LIN {X 0,Y 410.948,Z 878.716,A -85,B 0,C 180,E1 18093.627,E2 18093.627} C_VEL
LIN {X 0,Y 409.923,Z 893.274,A -85,B 0,C 180,E1 18092.657,E2 18092.657} C_VEL
LIN {X 0,Y 408.653,Z 907.82,A -85,B 0,C 180,E1 18091.402,E2 18091.402} C_VEL
LIN {X 0,Y 407.32,Z 921.375,A -85,B 0,C 180,E1 18089.93,E2 18089.93} C_VEL
LIN {X 0,Y 406.014,Z 933.316,A -85,B 0,C 180,E1 18088.307,E2 18088.307} C_VEL
LIN {X 0,Y 404.726,Z 944.345,A -85,B 0,C 180,E1 18086.441,E2 18086.441} C_VEL
LIN {X 0,Y 403.633,Z 953.739,A -85,B 0,C 180,E1 18084.456,E2 18084.456} C_VEL
LIN {X 0,Y 402.724,Z 961.665,A -85,B 0,C 180,E1 18082.296,E2 18082.296} C_VEL
LIN {X 0,Y 402.061,Z 968.085,A -85,B 0,C 180,E1 18079.975,E2 18079.975} C_VEL
LIN {X 0,Y 401.649,Z 972.603,A -85,B 0,C 180,E1 18077.638,E2 18077.638} C_VEL
LIN {X 0,Y 401.427,Z 975.501,A -85,B 0,C 180,E1 18075.11,E2 18075.11} C_VEL
LIN {X 0,Y 401.407,Z 976.508,A -85,B 0,C 180,E1 18072.758,E2 18072.758} C_VEL
LIN {X 0,Y 401.558,Z 975.728,A -85,B 0,C 180,E1 18070.255,E2 18070.255} C_VEL
LIN {X 0,Y 401.936,Z 973.165,A -85,B 0,C 180,E1 18067.783,E2 18067.783} C_VEL
LIN {X 0,Y 402.51,Z 969.039,A -85,B 0,C 180,E1 18065.491,E2 18065.491} C_VEL
LIN {X 0,Y 403.373,Z 962.973,A -85,B 0,C 180,E1 18063.171,E2 18063.171} C_VEL
LIN {X 0,Y 404.499,Z 955.48,A -85,B 0,C 180,E1 18061.022,E2 18061.022} C_VEL
LIN {X 0,Y 405.852,Z 946.406,A -85,B 0,C 180,E1 18059.01,E2 18059.01} C_VEL
LIN {X 0,Y 407.46,Z 935.302,A -85,B 0,C 180,E1 18057.059,E2 18057.059} C_VEL
LIN {X 0,Y 409.093,Z 923.229,A -85,B 0,C 180,E1 18055.365,E2 18055.365} C_VEL
LIN {X 0,Y 410.738,Z 909.55,A -85,B 0,C 180,E1 18053.843,E2 18053.843} C_VEL
LIN {X 0,Y 412.221,Z 895.286,A -85,B 0,C 180,E1 18052.584,E2 18052.584} C_VEL
LIN {X 0,Y 413.472,Z 880.507,A -85,B 0,C 180,E1 18051.576,E2 18051.576} C_VEL
LIN {X 0,Y 414.481,Z 863.966,A -85,B 0,C 180,E1 18050.742,E2 18050.742} C_VEL
LIN {X 0,Y 415.114,Z 847.179,A -85,B 0,C 180,E1 18050.169,E2 18050.169} C_VEL
LIN {X 0,Y 417.861,Z 722.491,A -85,B 0,C 180,E1 18047.832,E2 18047.832} C_VEL
LIN {X 0,Y 411.801,Z 695.607,A -85,B 0,C 180,E1 18046.697,E2 18046.697} C_VEL
LIN {X 0,Y 414.81,Z 668.603,A -85,B 0,C 180,E1 18042.474,E2 18042.474} C_VEL
LIN {X 0,Y 414.66,Z 666.207,A -85,B 0,C 180,E1 18042.041,E2 18042.041} C_VEL
LIN {X 0,Y 410.898,Z 651.984,A -85,B 0,C 180,E1 18039.068,E2 18039.068} C_VEL
LIN {X 0,Y 406.79,Z 639.122,A -85,B 0,C 180,E1 18036.151,E2 18036.151} C_VEL
LIN {X 0,Y 402.415,Z 627.066,A -85,B 0,C 180,E1 18033.142,E2 18033.142} C_VEL
LIN {X 0,Y 401.514,Z 624.334,A -85,B 0,C 180,E1 18032.371,E2 18032.371} C_VEL
LIN {X 0,Y 401.502,Z 624.212,A -85,B 0,C 180,E1 18028.402,E2 18028.402} C_VEL
LIN {X 0,Y 401.498,Z 624.219,A -85,B 0,C 180,E1 18024.419,E2 18024.419} C_VEL
LIN {X 0,Y 401.497,Z 624.224,A -85,B 0,C 180,E1 18020.405,E2 18020.405} C_VEL
LIN {X 0,Y 401.498,Z 624.224,A -85,B 0,C 180,E1 18016.344,E2 18016.344} C_VEL
LIN {X 0,Y 401.501,Z 624.222,A -85,B 0,C 180,E1 18012.367,E2 18012.367} C_VEL
LIN {X 0,Y 401.501,Z 624.22,A -85,B 0,C 180,E1 18008.305,E2 18008.305} C_VEL
LIN {X 0,Y 401.491,Z 624.213,A -85,B 0,C 180,E1 18004.428,E2 18004.428} C_VEL
LIN {X 0,Y 401.485,Z 624.204,A -85,B 0,C 180,E1 18000.428,E2 18000.428} C_VEL
LIN {X 0,Y 401.482,Z 624.205,A -85,B 0,C 180,E1 17996.431,E2 17996.431} C_VEL
LIN {X 0,Y 401.486,Z 624.215,A -85,B 0,C 180,E1 17992.416,E2 17992.416} C_VEL
LIN {X 0,Y 401.494,Z 624.224,A -85,B 0,C 180,E1 17988.508,E2 17988.508} C_VEL
LIN {X 0,Y 401.5,Z 624.215,A -85,B 0,C 180,E1 17984.525,E2 17984.525} C_VEL
LIN {X 0,Y 401.5,Z 624.206,A -85,B 0,C 180,E1 17980.507,E2 17980.507} C_VEL
LIN {X 0,Y 401.501,Z 624.205,A -85,B 0,C 180,E1 17976.519,E2 17976.519} C_VEL
LIN {X 0,Y 401.501,Z 624.206,A -85,B 0,C 180,E1 17972.568,E2 17972.568} C_VEL
LIN {X 0,Y 401.5,Z 624.207,A -85,B 0,C 180,E1 17968.636,E2 17968.636} C_VEL
LIN {X 0,Y 401.486,Z 624.213,A -85,B 0,C 180,E1 17964.706,E2 17964.706} C_VEL
LIN {X 0,Y 401.479,Z 624.224,A -85,B 0,C 180,E1 17960.76,E2 17960.76} C_VEL
LIN {X 0,Y 401.478,Z 624.222,A -85,B 0,C 180,E1 17956.775,E2 17956.775} C_VEL
LIN {X 0,Y 401.58,Z 624.794,A -85,B 0,C 180,E1 17956.338,E2 17956.338} C_VEL
LIN {X 0,Y 406.93,Z 637.442,A -85,B 0,C 180,E1 17953.665,E2 17953.665} C_VEL
LIN {X 0,Y 412.612,Z 651.727,A -85,B 0,C 180,E1 17950.989,E2 17950.989} C_VEL
LIN {X 0,Y 417.899,Z 667.344,A -85,B 0,C 180,E1 17948.423,E2 17948.423} C_VEL
LIN {X 0,Y 419.949,Z 674.277,A -85,B 0,C 180,E1 17947.382,E2 17947.382} C_VEL
LIN {X 0,Y 416.011,Z 707.311,A -85,B 0,C 180,E1 17943.954,E2 17943.954} C_VEL
LIN {X 0,Y 419.913,Z 739.224,A -85,B 0,C 180,E1 17942.952,E2 17942.952} C_VEL
LIN {X 0,Y 415.985,Z 917.427,A -85,B 0,C 180,E1 17939.753,E2 17939.753} C_VEL
LIN {X 0,Y 414.846,Z 936.641,A -85,B 0,C 180,E1 17939.174,E2 17939.174} C_VEL
LIN {X 0,Y 413.402,Z 954.824,A -85,B 0,C 180,E1 17938.376,E2 17938.376} C_VEL
LIN {X 0,Y 411.674,Z 972.774,A -85,B 0,C 180,E1 17937.325,E2 17937.325} C_VEL
LIN {X 0,Y 409.84,Z 989.883,A -85,B 0,C 180,E1 17936.048,E2 17936.048} C_VEL
LIN {X 0,Y 407.953,Z 1006.197,A -85,B 0,C 180,E1 17934.546,E2 17934.546} C_VEL
LIN {X 0,Y 406.111,Z 1021.663,A -85,B 0,C 180,E1 17932.815,E2 17932.815} C_VEL
LIN {X 0,Y 404.421,Z 1036.236,A -85,B 0,C 180,E1 17930.847,E2 17930.847} C_VEL
LIN {X 0,Y 402.954,Z 1049.621,A -85,B 0,C 180,E1 17928.668,E2 17928.668} C_VEL
LIN {X 0,Y 401.838,Z 1061.521,A -85,B 0,C 180,E1 17926.33,E2 17926.33} C_VEL
LIN {X 0,Y 401.058,Z 1071.88,A -85,B 0,C 180,E1 17923.847,E2 17923.847} C_VEL
LIN {X 0,Y 400.626,Z 1080.6,A -85,B 0,C 180,E1 17921.239,E2 17921.239} C_VEL
LIN {X 0,Y 400.459,Z 1087.386,A -85,B 0,C 180,E1 17918.613,E2 17918.613} C_VEL
LIN {X 0,Y 400.468,Z 1092.26,A -85,B 0,C 180,E1 17916.019,E2 17916.019} C_VEL
LIN {X 0,Y 400.552,Z 1095.388,A -85,B 0,C 180,E1 17913.434,E2 17913.434} C_VEL
LIN {X 0,Y 400.609,Z 1096.821,A -85,B 0,C 180,E1 17910.858,E2 17910.858} C_VEL
LIN {X 0,Y 400.591,Z 1096.647,A -85,B 0,C 180,E1 17908.426,E2 17908.426} C_VEL
LIN {X 0,Y 400.513,Z 1094.819,A -85,B 0,C 180,E1 17905.848,E2 17905.848} C_VEL
LIN {X 0,Y 400.431,Z 1091.265,A -85,B 0,C 180,E1 17903.26,E2 17903.26} C_VEL
LIN {X 0,Y 400.461,Z 1085.91,A -85,B 0,C 180,E1 17900.66,E2 17900.66} C_VEL
LIN {X 0,Y 400.699,Z 1078.507,A -85,B 0,C 180,E1 17898.001,E2 17898.001} C_VEL
LIN {X 0,Y 401.246,Z 1069.273,A -85,B 0,C 180,E1 17895.423,E2 17895.423} C_VEL
LIN {X 0,Y 402.084,Z 1058.931,A -85,B 0,C 180,E1 17893.085,E2 17893.085} C_VEL
LIN {X 0,Y 403.252,Z 1046.965,A -85,B 0,C 180,E1 17890.854,E2 17890.854} C_VEL
LIN {X 0,Y 404.735,Z 1033.331,A -85,B 0,C 180,E1 17888.749,E2 17888.749} C_VEL
LIN {X 0,Y 406.383,Z 1018.854,A -85,B 0,C 180,E1 17886.894,E2 17886.894} C_VEL
LIN {X 0,Y 408.163,Z 1003.233,A -85,B 0,C 180,E1 17885.235,E2 17885.235} C_VEL
LIN {X 0,Y 409.958,Z 986.785,A -85,B 0,C 180,E1 17883.803,E2 17883.803} C_VEL
LIN {X 0,Y 411.678,Z 969.565,A -85,B 0,C 180,E1 17882.597,E2 17882.597} C_VEL
LIN {X 0,Y 413.244,Z 951.519,A -85,B 0,C 180,E1 17881.612,E2 17881.612} C_VEL
LIN {X 0,Y 414.584,Z 932.755,A -85,B 0,C 180,E1 17880.86,E2 17880.86} C_VEL
LIN {X 0,Y 415.491,Z 913.481,A -85,B 0,C 180,E1 17880.346,E2 17880.346} C_VEL
LIN {X 0,Y 418.723,Z 737.102,A -85,B 0,C 180,E1 17877.259,E2 17877.259} C_VEL
LIN {X 0,Y 414.963,Z 707.158,A -85,B 0,C 180,E1 17876.389,E2 17876.389} C_VEL
LIN {X 0,Y 418.463,Z 672.256,A -85,B 0,C 180,E1 17872.887,E2 17872.887} C_VEL
LIN {X 0,Y 411.146,Z 650.69,A -85,B 0,C 180,E1 17869.783,E2 17869.783} C_VEL
LIN {X 0,Y 403.769,Z 630.541,A -85,B 0,C 180,E1 17866.618,E2 17866.618} C_VEL
LIN {X 0,Y 401.517,Z 624.406,A -85,B 0,C 180,E1 17865.527,E2 17865.527} C_VEL
LIN {X 0,Y 401.497,Z 624.217,A -85,B 0,C 180,E1 17861.66,E2 17861.66} C_VEL
LIN {X 0,Y 401.499,Z 624.222,A -85,B 0,C 180,E1 17857.779,E2 17857.779} C_VEL
LIN {X 0,Y 401.492,Z 624.224,A -85,B 0,C 180,E1 17853.906,E2 17853.906} C_VEL
LIN {X 0,Y 401.484,Z 624.224,A -85,B 0,C 180,E1 17849.926,E2 17849.926} C_VEL
LIN {X 0,Y 401.483,Z 624.224,A -85,B 0,C 180,E1 17845.967,E2 17845.967} C_VEL
LIN {X 0,Y 401.488,Z 624.225,A -85,B 0,C 180,E1 17842.089,E2 17842.089} C_VEL
LIN {X 0,Y 401.49,Z 624.226,A -85,B 0,C 180,E1 17838.137,E2 17838.137} C_VEL
LIN {X 0,Y 401.509,Z 624.334,A -85,B 0,C 180,E1 17834.714,E2 17834.714} C_VEL
LIN {X 0,Y 402.009,Z 626.178,A -85,B 0,C 180,E1 17834.328,E2 17834.328} C_VEL
LIN {X 0,Y 406.281,Z 636.393,A -85,B 0,C 180,E1 17832.58,E2 17832.58} C_VEL
LIN {X 0,Y 410.796,Z 649.556,A -85,B 0,C 180,E1 17830.518,E2 17830.518} C_VEL
LIN {X 0,Y 413.885,Z 662.108,A -85,B 0,C 180,E1 17828.684,E2 17828.684} C_VEL
LIN {X 0,Y 413.166,Z 694.495,A -85,B 0,C 180,E1 17824.859,E2 17824.859} C_VEL
LIN {X 0,Y 412.587,Z 720.52,A -85,B 0,C 180,E1 17821.757,E2 17821.757} C_VEL
LIN {X 0,Y 412.786,Z 724.532,A -85,B 0,C 180,E1 17821.644,E2 17821.644} C_VEL
LIN {X 0,Y 409.599,Z 849.624,A -85,B 0,C 180,E1 17819.025,E2 17819.025} C_VEL
LIN {X 0,Y 409.503,Z 867.341,A -85,B 0,C 180,E1 17818.522,E2 17818.522} C_VEL
LIN {X 0,Y 409.073,Z 883.957,A -85,B 0,C 180,E1 17817.758,E2 17817.758} C_VEL
LIN {X 0,Y 408.449,Z 898.379,A -85,B 0,C 180,E1 17816.842,E2 17816.842} C_VEL
LIN {X 0,Y 407.57,Z 912.742,A -85,B 0,C 180,E1 17815.638,E2 17815.638} C_VEL
LIN {X 0,Y 406.631,Z 925.44,A -85,B 0,C 180,E1 17814.284,E2 17814.284} C_VEL
LIN {X 0,Y 405.541,Z 937.675,A -85,B 0,C 180,E1 17812.634,E2 17812.634} C_VEL
LIN {X 0,Y 404.547,Z 947.904,A -85,B 0,C 180,E1 17810.898,E2 17810.898} C_VEL
LIN {X 0,Y 403.573,Z 957.408,A -85,B 0,C 180,E1 17808.844,E2 17808.844} C_VEL
LIN {X 0,Y 402.819,Z 964.607,A -85,B 0,C 180,E1 17806.799,E2 17806.799} C_VEL
LIN {X 0,Y 402.216,Z 970.369,A -85,B 0,C 180,E1 17804.574,E2 17804.574} C_VEL
LIN {X 0,Y 401.791,Z 974.195,A -85,B 0,C 180,E1 17802.326,E2 17802.326} C_VEL
LIN {X 0,Y 401.543,Z 976.273,A -85,B 0,C 180,E1 17800.054,E2 17800.054} C_VEL
LIN {X 0,Y 401.425,Z 976.558,A -85,B 0,C 180,E1 17797.753,E2 17797.753} C_VEL
LIN {X 0,Y 401.434,Z 975.029,A -85,B 0,C 180,E1 17795.384,E2 17795.384} C_VEL
LIN {X 0,Y 401.568,Z 971.912,A -85,B 0,C 180,E1 17793.213,E2 17793.213} C_VEL
LIN {X 0,Y 401.869,Z 966.938,A -85,B 0,C 180,E1 17790.976,E2 17790.976} C_VEL
LIN {X 0,Y 402.325,Z 960.411,A -85,B 0,C 180,E1 17788.874,E2 17788.874} C_VEL
LIN {X 0,Y 402.989,Z 951.677,A -85,B 0,C 180,E1 17786.735,E2 17786.735} C_VEL
LIN {X 0,Y 403.732,Z 942.257,A -85,B 0,C 180,E1 17784.931,E2 17784.931} C_VEL
LIN {X 0,Y 404.673,Z 930.317,A -85,B 0,C 180,E1 17783.101,E2 17783.101} C_VEL
LIN {X 0,Y 405.573,Z 917.892,A -85,B 0,C 180,E1 17781.592,E2 17781.592} C_VEL
LIN {X 0,Y 406.458,Z 904.008,A -85,B 0,C 180,E1 17780.239,E2 17780.239} C_VEL
LIN {X 0,Y 407.25,Z 888.689,A -85,B 0,C 180,E1 17779.089,E2 17779.089} C_VEL
LIN {X 0,Y 407.854,Z 873.417,A -85,B 0,C 180,E1 17778.225,E2 17778.225} C_VEL
LIN {X 0,Y 408.225,Z 856.157,A -85,B 0,C 180,E1 17777.554,E2 17777.554} C_VEL
LIN {X 0,Y 408.39,Z 834.696,A -85,B 0,C 180,E1 17777.069,E2 17777.069} C_VEL
LIN {X 0,Y 410.575,Z 718.657,A -85,B 0,C 180,E1 17774.8,E2 17774.8} C_VEL
LIN {X 0,Y 409.2,Z 710.904,A -85,B 0,C 180,E1 17774.53,E2 17774.53} C_VEL
LIN {X 0,Y 410.192,Z 680.126,A -85,B 0,C 180,E1 17770.705,E2 17770.705} C_VEL
LIN {X 0,Y 410.726,Z 657.174,A -85,B 0,C 180,E1 17767.841,E2 17767.841} C_VEL
LIN {X 0,Y 405.666,Z 638.159,A -85,B 0,C 180,E1 17765.05,E2 17765.05} C_VEL
LIN {X 0,Y 401.475,Z 624.396,A -85,B 0,C 180,E1 17762.912,E2 17762.912} C_VEL
LIN {X 0,Y 401.489,Z 624.225,A -85,B 0,C 180,E1 17761.35,E2 17761.35} C_VEL
LIN {X 0,Y 400.432,Z 624.354,A -85,B 0,C 180,E1 17760.251,E2 17760.251} C_VEL
LIN {X 0,Y 393.938,Z 625.162,A -85,B 0,C 180,E1 17757.072,E2 17757.072} C_VEL
LIN {X 0,Y 393.509,Z 625.198,A -85,B 0,C 180,E1 17756.342,E2 17756.342} C_VEL
LIN {X 0,Y 393.515,Z 625.213,A -85,B 0,C 180,E1 17752.351,E2 17752.351} C_VEL
LIN {X 0,Y 393.611,Z 625.529,A -85,B 0,C 180,E1 17751.144,E2 17751.144} C_VEL
LIN {X 0,Y 398.734,Z 642.233,A -85,B 0,C 180,E1 17747.657,E2 17747.657} C_VEL
LIN {X 0,Y 403.375,Z 659.305,A -85,B 0,C 180,E1 17744.352,E2 17744.352} C_VEL
LIN {X 0,Y 404.657,Z 665.567,A -85,B 0,C 180,E1 17743.211,E2 17743.211} C_VEL
LIN {X 0,Y 401.936,Z 693.579,A -85,B 0,C 180,E1 17738.873,E2 17738.873} C_VEL
LIN {X 0,Y 401.915,Z 695.836,A -85,B 0,C 180,E1 17738.621,E2 17738.621} C_VEL
LIN {X 0,Y 407.444,Z 724.144,A -85,B 0,C 180,E1 17737.677,E2 17737.677} C_VEL
LIN {X 0,Y 404.979,Z 846.669,A -85,B 0,C 180,E1 17735.424,E2 17735.424} C_VEL
LIN {X 0,Y 404.395,Z 863.875,A -85,B 0,C 180,E1 17734.831,E2 17734.831} C_VEL
LIN {X 0,Y 403.562,Z 879.387,A -85,B 0,C 180,E1 17734.049,E2 17734.049} C_VEL
LIN {X 0,Y 402.492,Z 894.012,A -85,B 0,C 180,E1 17733.062,E2 17733.062} C_VEL
LIN {X 0,Y 401.135,Z 908.873,A -85,B 0,C 180,E1 17731.759,E2 17731.759} C_VEL
LIN {X 0,Y 399.76,Z 922.197,A -85,B 0,C 180,E1 17730.287,E2 17730.287} C_VEL
LIN {X 0,Y 398.444,Z 933.729,A -85,B 0,C 180,E1 17728.706,E2 17728.706} C_VEL
LIN {X 0,Y 397.085,Z 944.773,A -85,B 0,C 180,E1 17726.825,E2 17726.825} C_VEL
LIN {X 0,Y 395.904,Z 954.369,A -85,B 0,C 180,E1 17724.784,E2 17724.784} C_VEL
LIN {X 0,Y 394.99,Z 961.973,A -85,B 0,C 180,E1 17722.729,E2 17722.729} C_VEL
LIN {X 0,Y 394.252,Z 968.582,A -85,B 0,C 180,E1 17720.365,E2 17720.365} C_VEL
LIN {X 0,Y 393.789,Z 973.345,A -85,B 0,C 180,E1 17717.983,E2 17717.983} C_VEL
LIN {X 0,Y 393.539,Z 976.31,A -85,B 0,C 180,E1 17715.583,E2 17715.583} C_VEL
LIN {X 0,Y 393.487,Z 977.642,A -85,B 0,C 180,E1 17713.01,E2 17713.01} C_VEL
LIN {X 0,Y 393.631,Z 977.211,A -85,B 0,C 180,E1 17710.564,E2 17710.564} C_VEL
LIN {X 0,Y 393.986,Z 974.982,A -85,B 0,C 180,E1 17708.096,E2 17708.096} C_VEL
LIN {X 0,Y 394.603,Z 970.926,A -85,B 0,C 180,E1 17705.606,E2 17705.606} C_VEL
LIN {X 0,Y 395.488,Z 965.214,A -85,B 0,C 180,E1 17703.256,E2 17703.256} C_VEL
LIN {X 0,Y 396.743,Z 957.38,A -85,B 0,C 180,E1 17700.897,E2 17700.897} C_VEL
LIN {X 0,Y 398.171,Z 948.589,A -85,B 0,C 180,E1 17698.85,E2 17698.85} C_VEL
LIN {X 0,Y 399.806,Z 937.996,A -85,B 0,C 180,E1 17696.908,E2 17696.908} C_VEL
LIN {X 0,Y 401.524,Z 926.181,A -85,B 0,C 180,E1 17695.169,E2 17695.169} C_VEL
LIN {X 0,Y 403.213,Z 913.39,A -85,B 0,C 180,E1 17693.655,E2 17693.655} C_VEL
LIN {X 0,Y 404.818,Z 899.074,A -85,B 0,C 180,E1 17692.317,E2 17692.317} C_VEL
LIN {X 0,Y 406.277,Z 883.536,A -85,B 0,C 180,E1 17691.187,E2 17691.187} C_VEL
LIN {X 0,Y 407.372,Z 867.647,A -85,B 0,C 180,E1 17690.329,E2 17690.329} C_VEL
LIN {X 0,Y 408.106,Z 850.469,A -85,B 0,C 180,E1 17689.693,E2 17689.693} C_VEL
LIN {X 0,Y 408.732,Z 823.466,A -85,B 0,C 180,E1 17689.121,E2 17689.121} C_VEL
LIN {X 0,Y 411.102,Z 723.877,A -85,B 0,C 180,E1 17687.253,E2 17687.253} C_VEL
LIN {X 0,Y 404.768,Z 695.985,A -85,B 0,C 180,E1 17686.043,E2 17686.043} C_VEL
LIN {X 0,Y 407.748,Z 670.492,A -85,B 0,C 180,E1 17682.013,E2 17682.013} C_VEL
LIN {X 0,Y 404.253,Z 656.746,A -85,B 0,C 180,E1 17679.103,E2 17679.103} C_VEL
LIN {X 0,Y 400.252,Z 643.813,A -85,B 0,C 180,E1 17676.125,E2 17676.125} C_VEL
LIN {X 0,Y 395.853,Z 631.559,A -85,B 0,C 180,E1 17673.01,E2 17673.01} C_VEL
LIN {X 0,Y 393.578,Z 625.315,A -85,B 0,C 180,E1 17671.253,E2 17671.253} C_VEL
LIN {X 0,Y 393.565,Z 625.213,A -85,B 0,C 180,E1 17667.213,E2 17667.213} C_VEL
LIN {X 0,Y 393.561,Z 625.205,A -85,B 0,C 180,E1 17663.122,E2 17663.122} C_VEL
LIN {X 0,Y 393.556,Z 625.199,A -85,B 0,C 180,E1 17659.075,E2 17659.075} C_VEL
LIN {X 0,Y 393.549,Z 625.199,A -85,B 0,C 180,E1 17655.109,E2 17655.109} C_VEL
LIN {X 0,Y 393.55,Z 625.202,A -85,B 0,C 180,E1 17651.133,E2 17651.133} C_VEL
LIN {X 0,Y 393.555,Z 625.208,A -85,B 0,C 180,E1 17647.152,E2 17647.152} C_VEL
LIN {X 0,Y 393.557,Z 625.214,A -85,B 0,C 180,E1 17643.201,E2 17643.201} C_VEL
LIN {X 0,Y 393.562,Z 625.203,A -85,B 0,C 180,E1 17639.127,E2 17639.127} C_VEL
LIN {X 0,Y 393.558,Z 625.19,A -85,B 0,C 180,E1 17635.045,E2 17635.045} C_VEL
LIN {X 0,Y 393.559,Z 625.189,A -85,B 0,C 180,E1 17631.085,E2 17631.085} C_VEL
LIN {X 0,Y 393.56,Z 625.198,A -85,B 0,C 180,E1 17627.082,E2 17627.082} C_VEL
LIN {X 0,Y 393.562,Z 625.211,A -85,B 0,C 180,E1 17623.165,E2 17623.165} C_VEL
LIN {X 0,Y 393.56,Z 625.211,A -85,B 0,C 180,E1 17619.165,E2 17619.165} C_VEL
LIN {X 0,Y 393.549,Z 625.212,A -85,B 0,C 180,E1 17615.216,E2 17615.216} C_VEL
LIN {X 0,Y 393.545,Z 625.211,A -85,B 0,C 180,E1 17611.225,E2 17611.225} C_VEL
LIN {X 0,Y 393.543,Z 625.214,A -85,B 0,C 180,E1 17607.238,E2 17607.238} C_VEL
LIN {X 0,Y 393.547,Z 625.214,A -85,B 0,C 180,E1 17603.341,E2 17603.341} C_VEL
LIN {X 0,Y 393.561,Z 625.203,A -85,B 0,C 180,E1 17599.43,E2 17599.43} C_VEL
LIN {X 0,Y 393.6,Z 625.474,A -85,B 0,C 180,E1 17597.551,E2 17597.551} C_VEL
LIN {X 0,Y 398.76,Z 637.635,A -85,B 0,C 180,E1 17594.796,E2 17594.796} C_VEL
LIN {X 0,Y 404.277,Z 651.337,A -85,B 0,C 180,E1 17592.085,E2 17592.085} C_VEL
LIN {X 0,Y 409.518,Z 666.021,A -85,B 0,C 180,E1 17589.509,E2 17589.509} C_VEL
LIN {X 0,Y 412.843,Z 677.235,A -85,B 0,C 180,E1 17587.743,E2 17587.743} C_VEL
LIN {X 0,Y 409.049,Z 707.569,A -85,B 0,C 180,E1 17584.547,E2 17584.547} C_VEL
LIN {X 0,Y 413.042,Z 740.309,A -85,B 0,C 180,E1 17583.504,E2 17583.504} C_VEL
LIN {X 0,Y 408.913,Z 916.579,A -85,B 0,C 180,E1 17580.285,E2 17580.285} C_VEL
LIN {X 0,Y 407.728,Z 935.734,A -85,B 0,C 180,E1 17579.699,E2 17579.699} C_VEL
LIN {X 0,Y 406.253,Z 953.317,A -85,B 0,C 180,E1 17578.922,E2 17578.922} C_VEL
LIN {X 0,Y 404.435,Z 971.385,A -85,B 0,C 180,E1 17577.856,E2 17577.856} C_VEL
LIN {X 0,Y 402.486,Z 988.565,A -85,B 0,C 180,E1 17576.561,E2 17576.561} C_VEL
LIN {X 0,Y 400.472,Z 1004.977,A -85,B 0,C 180,E1 17575.028,E2 17575.028} C_VEL
LIN {X 0,Y 398.525,Z 1020.37,A -85,B 0,C 180,E1 17573.275,E2 17573.275} C_VEL
LIN {X 0,Y 396.728,Z 1034.89,A -85,B 0,C 180,E1 17571.279,E2 17571.279} C_VEL
LIN {X 0,Y 395.252,Z 1047.548,A -85,B 0,C 180,E1 17569.199,E2 17569.199} C_VEL
LIN {X 0,Y 394.023,Z 1059.595,A -85,B 0,C 180,E1 17566.815,E2 17566.815} C_VEL
LIN {X 0,Y 393.162,Z 1070.08,A -85,B 0,C 180,E1 17564.281,E2 17564.281} C_VEL
LIN {X 0,Y 392.68,Z 1078.97,A -85,B 0,C 180,E1 17561.604,E2 17561.604} C_VEL
LIN {X 0,Y 392.504,Z 1085.837,A -85,B 0,C 180,E1 17558.939,E2 17558.939} C_VEL
LIN {X 0,Y 392.519,Z 1090.833,A -85,B 0,C 180,E1 17556.288,E2 17556.288} C_VEL
LIN {X 0,Y 392.622,Z 1094.07,A -85,B 0,C 180,E1 17553.65,E2 17553.65} C_VEL
LIN {X 0,Y 392.694,Z 1095.604,A -85,B 0,C 180,E1 17551.021,E2 17551.021} C_VEL
LIN {X 0,Y 392.678,Z 1095.522,A -85,B 0,C 180,E1 17548.541,E2 17548.541} C_VEL
LIN {X 0,Y 392.59,Z 1093.764,A -85,B 0,C 180,E1 17545.91,E2 17545.91} C_VEL
LIN {X 0,Y 392.492,Z 1090.261,A -85,B 0,C 180,E1 17543.27,E2 17543.27} C_VEL
LIN {X 0,Y 392.504,Z 1084.969,A -85,B 0,C 180,E1 17540.617,E2 17540.617} C_VEL
LIN {X 0,Y 392.707,Z 1078.215,A -85,B 0,C 180,E1 17538.098,E2 17538.098} C_VEL
LIN {X 0,Y 393.204,Z 1069.612,A -85,B 0,C 180,E1 17535.569,E2 17535.569} C_VEL
LIN {X 0,Y 394.026,Z 1059.571,A -85,B 0,C 180,E1 17533.185,E2 17533.185} C_VEL
LIN {X 0,Y 395.163,Z 1048.166,A -85,B 0,C 180,E1 17530.949,E2 17530.949} C_VEL
LIN {X 0,Y 396.657,Z 1034.941,A -85,B 0,C 180,E1 17528.794,E2 17528.794} C_VEL
LIN {X 0,Y 398.417,Z 1020.149,A -85,B 0,C 180,E1 17526.796,E2 17526.796} C_VEL
LIN {X 0,Y 400.323,Z 1004.299,A -85,B 0,C 180,E1 17525.032,E2 17525.032} C_VEL
LIN {X 0,Y 402.243,Z 987.624,A -85,B 0,C 180,E1 17523.522,E2 17523.522} C_VEL
LIN {X 0,Y 404.046,Z 970.475,A -85,B 0,C 180,E1 17522.275,E2 17522.275} C_VEL
LIN {X 0,Y 405.725,Z 952.163,A -85,B 0,C 180,E1 17521.238,E2 17521.238} C_VEL
LIN {X 0,Y 407.153,Z 933.246,A -85,B 0,C 180,E1 17520.451,E2 17520.451} C_VEL
LIN {X 0,Y 408.129,Z 914.052,A -85,B 0,C 180,E1 17519.916,E2 17519.916} C_VEL
LIN {X 0,Y 411.541,Z 738.121,A -85,B 0,C 180,E1 17516.783,E2 17516.783} C_VEL
LIN {X 0,Y 407.676,Z 707.337,A -85,B 0,C 180,E1 17515.894,E2 17515.894} C_VEL
LIN {X 0,Y 411.164,Z 675.114,A -85,B 0,C 180,E1 17512.607,E2 17512.607} C_VEL
LIN {X 0,Y 404.132,Z 654.184,A -85,B 0,C 180,E1 17509.544,E2 17509.544} C_VEL
LIN {X 0,Y 397.156,Z 634.971,A -85,B 0,C 180,E1 17506.473,E2 17506.473} C_VEL
LIN {X 0,Y 393.584,Z 625.393,A -85,B 0,C 180,E1 17504.766,E2 17504.766} C_VEL
LIN {X 0,Y 393.567,Z 625.208,A -85,B 0,C 180,E1 17500.761,E2 17500.761} C_VEL
LIN {X 0,Y 393.561,Z 625.211,A -85,B 0,C 180,E1 17496.839,E2 17496.839} C_VEL
LIN {X 0,Y 393.56,Z 625.211,A -85,B 0,C 180,E1 17492.761,E2 17492.761} C_VEL
LIN {X 0,Y 393.569,Z 625.212,A -85,B 0,C 180,E1 17488.695,E2 17488.695} C_VEL
LIN {X 0,Y 393.566,Z 625.211,A -85,B 0,C 180,E1 17484.623,E2 17484.623} C_VEL
LIN {X 0,Y 393.569,Z 625.212,A -85,B 0,C 180,E1 17480.679,E2 17480.679} C_VEL
LIN {X 0,Y 393.561,Z 625.213,A -85,B 0,C 180,E1 17476.683,E2 17476.683} C_VEL
LIN {X 0,Y 393.565,Z 625.482,A -85,B 0,C 180,E1 17475.622,E2 17475.622} C_VEL
LIN {X 0,Y 394.9,Z 628.784,A -85,B 0,C 180,E1 17474.966,E2 17474.966} C_VEL
LIN {X 0,Y 400.239,Z 641.697,A -85,B 0,C 180,E1 17472.699,E2 17472.699} C_VEL
LIN {X 0,Y 404.726,Z 655.471,A -85,B 0,C 180,E1 17470.501,E2 17470.501} C_VEL
LIN {X 0,Y 406.969,Z 665.302,A -85,B 0,C 180,E1 17469.046,E2 17469.046} C_VEL
LIN {X 0,Y 406.169,Z 696.789,A -85,B 0,C 180,E1 17465.296,E2 17465.296} C_VEL
LIN {X 0,Y 405.53,Z 721.985,A -85,B 0,C 180,E1 17462.269,E2 17462.269} C_VEL
LIN {X 0,Y 405.725,Z 725.942,A -85,B 0,C 180,E1 17462.154,E2 17462.154} C_VEL
LIN {X 0,Y 402.305,Z 847.525,A -85,B 0,C 180,E1 17459.537,E2 17459.537} C_VEL
LIN {X 0,Y 402.217,Z 866.083,A -85,B 0,C 180,E1 17459.038,E2 17459.038} C_VEL
LIN {X 0,Y 401.86,Z 881.788,A -85,B 0,C 180,E1 17458.36,E2 17458.36} C_VEL
LIN {X 0,Y 401.192,Z 896.972,A -85,B 0,C 180,E1 17457.429,E2 17457.429} C_VEL
LIN {X 0,Y 400.326,Z 911.218,A -85,B 0,C 180,E1 17456.276,E2 17456.276} C_VEL
LIN {X 0,Y 399.259,Z 925.079,A -85,B 0,C 180,E1 17454.827,E2 17454.827} C_VEL
LIN {X 0,Y 398.245,Z 936.232,A -85,B 0,C 180,E1 17453.368,E2 17453.368} C_VEL
LIN {X 0,Y 397.141,Z 946.99,A -85,B 0,C 180,E1 17451.603,E2 17451.603} C_VEL
LIN {X 0,Y 396.127,Z 956.316,A -85,B 0,C 180,E1 17449.676,E2 17449.676} C_VEL
LIN {X 0,Y 395.235,Z 964.19,A -85,B 0,C 180,E1 17447.556,E2 17447.556} C_VEL
LIN {X 0,Y 394.578,Z 970.034,A -85,B 0,C 180,E1 17445.465,E2 17445.465} C_VEL
LIN {X 0,Y 394.052,Z 974.431,A -85,B 0,C 180,E1 17443.186,E2 17443.186} C_VEL
LIN {X 0,Y 393.724,Z 977.083,A -85,B 0,C 180,E1 17440.856,E2 17440.856} C_VEL
LIN {X 0,Y 393.544,Z 977.893,A -85,B 0,C 180,E1 17438.417,E2 17438.417} C_VEL
LIN {X 0,Y 393.508,Z 976.962,A -85,B 0,C 180,E1 17436.167,E2 17436.167} C_VEL
LIN {X 0,Y 393.612,Z 974.05,A -85,B 0,C 180,E1 17433.728,E2 17433.728} C_VEL
LIN {X 0,Y 393.886,Z 969.49,A -85,B 0,C 180,E1 17431.439,E2 17431.439} C_VEL
LIN {X 0,Y 394.345,Z 963.075,A -85,B 0,C 180,E1 17429.191,E2 17429.191} C_VEL
LIN {X 0,Y 394.928,Z 955.554,A -85,B 0,C 180,E1 17427.194,E2 17427.194} C_VEL
LIN {X 0,Y 395.764,Z 945.394,A -85,B 0,C 180,E1 17425.094,E2 17425.094} C_VEL
LIN {X 0,Y 396.657,Z 934.498,A -85,B 0,C 180,E1 17423.315,E2 17423.315} C_VEL
LIN {X 0,Y 397.679,Z 921.432,A -85,B 0,C 180,E1 17421.609,E2 17421.609} C_VEL
LIN {X 0,Y 398.576,Z 908.058,A -85,B 0,C 180,E1 17420.231,E2 17420.231} C_VEL
LIN {X 0,Y 399.44,Z 893.131,A -85,B 0,C 180,E1 17419.017,E2 17419.017} C_VEL
LIN {X 0,Y 400.124,Z 877.239,A -85,B 0,C 180,E1 17418.052,E2 17418.052} C_VEL
LIN {X 0,Y 400.56,Z 861.087,A -85,B 0,C 180,E1 17417.352,E2 17417.352} C_VEL
LIN {X 0,Y 400.731,Z 842.468,A -85,B 0,C 180,E1 17416.863,E2 17416.863} C_VEL
LIN {X 0,Y 403.114,Z 719.67,A -85,B 0,C 180,E1 17414.398,E2 17414.398} C_VEL
LIN {X 0,Y 401.725,Z 711.979,A -85,B 0,C 180,E1 17414.137,E2 17414.137} C_VEL
LIN {X 0,Y 402.764,Z 681.31,A -85,B 0,C 180,E1 17410.302,E2 17410.302} C_VEL
LIN {X 0,Y 403.271,Z 659.615,A -85,B 0,C 180,E1 17407.585,E2 17407.585} C_VEL
LIN {X 0,Y 398.366,Z 641.115,A -85,B 0,C 180,E1 17404.841,E2 17404.841} C_VEL
LIN {X 0,Y 393.534,Z 625.4,A -85,B 0,C 180,E1 17402.377,E2 17402.377} C_VEL
LIN {X 0,Y 393.51,Z 625.214,A -85,B 0,C 180,E1 17398.369,E2 17398.369} C_VEL
LIN {X 0,Y 393.509,Z 625.198,A -85,B 0,C 180,E1 17396.342,E2 17396.342} C_VEL
LIN {X 0,Y 392.526,Z 625.305,A -85,B 0,C 180,E1 17395.597,E2 17395.597} C_VEL
LIN {X 0,Y 386.187,Z 626.094,A -85,B 0,C 180,E1 17393.564,E2 17393.564} C_VEL
LIN {X 0,Y 385.613,Z 626.176,A -85,B 0,C 180,E1 17393.011,E2 17393.011} C_VEL
LIN {X 0,Y 385.631,Z 626.546,A -85,B 0,C 180,E1 17391.871,E2 17391.871} C_VEL
LIN {X 0,Y 390.356,Z 641.681,A -85,B 0,C 180,E1 17388.607,E2 17388.607} C_VEL
LIN {X 0,Y 394.773,Z 657.568,A -85,B 0,C 180,E1 17385.423,E2 17385.423} C_VEL
LIN {X 0,Y 397.239,Z 667.51,A -85,B 0,C 180,E1 17383.538,E2 17383.538} C_VEL
LIN {X 0,Y 394.473,Z 695.115,A -85,B 0,C 180,E1 17379.226,E2 17379.226} C_VEL
LIN {X 0,Y 395.815,Z 702.455,A -85,B 0,C 180,E1 17378.927,E2 17378.927} C_VEL
LIN {X 0,Y 400.244,Z 725.47,A -85,B 0,C 180,E1 17378.157,E2 17378.157} C_VEL
LIN {X 0,Y 397.669,Z 847.208,A -85,B 0,C 180,E1 17375.881,E2 17375.881} C_VEL
LIN {X 0,Y 397.062,Z 864.382,A -85,B 0,C 180,E1 17375.283,E2 17375.283} C_VEL
LIN {X 0,Y 396.131,Z 880.962,A -85,B 0,C 180,E1 17374.43,E2 17374.43} C_VEL
LIN {X 0,Y 394.909,Z 896.445,A -85,B 0,C 180,E1 17373.339,E2 17373.339} C_VEL
LIN {X 0,Y 393.46,Z 911.489,A -85,B 0,C 180,E1 17371.966,E2 17371.966} C_VEL
LIN {X 0,Y 392.011,Z 924.697,A -85,B 0,C 180,E1 17370.439,E2 17370.439} C_VEL
LIN {X 0,Y 390.53,Z 936.856,A -85,B 0,C 180,E1 17368.68,E2 17368.68} C_VEL
LIN {X 0,Y 389.156,Z 947.566,A -85,B 0,C 180,E1 17366.76,E2 17366.76} C_VEL
LIN {X 0,Y 387.953,Z 956.795,A -85,B 0,C 180,E1 17364.677,E2 17364.677} C_VEL
LIN {X 0,Y 386.978,Z 964.561,A -85,B 0,C 180,E1 17362.428,E2 17362.428} C_VEL
LIN {X 0,Y 386.264,Z 970.848,A -85,B 0,C 180,E1 17360.013,E2 17360.013} C_VEL
LIN {X 0,Y 385.819,Z 975.205,A -85,B 0,C 180,E1 17357.579,E2 17357.579} C_VEL
LIN {X 0,Y 385.596,Z 977.992,A -85,B 0,C 180,E1 17354.972,E2 17354.972} C_VEL
LIN {X 0,Y 385.592,Z 978.899,A -85,B 0,C 180,E1 17352.495,E2 17352.495} C_VEL
LIN {X 0,Y 385.807,Z 978.005,A -85,B 0,C 180,E1 17349.838,E2 17349.838} C_VEL
LIN {X 0,Y 386.267,Z 975.409,A -85,B 0,C 180,E1 17347.314,E2 17347.314} C_VEL
LIN {X 0,Y 386.958,Z 971.187,A -85,B 0,C 180,E1 17344.928,E2 17344.928} C_VEL
LIN {X 0,Y 388.04,Z 964.798,A -85,B 0,C 180,E1 17342.423,E2 17342.423} C_VEL
LIN {X 0,Y 389.349,Z 957.292,A -85,B 0,C 180,E1 17340.227,E2 17340.227} C_VEL
LIN {X 0,Y 390.939,Z 947.969,A -85,B 0,C 180,E1 17338.117,E2 17338.117} C_VEL
LIN {X 0,Y 392.769,Z 936.863,A -85,B 0,C 180,E1 17336.117,E2 17336.117} C_VEL
LIN {X 0,Y 394.542,Z 925.202,A -85,B 0,C 180,E1 17334.439,E2 17334.439} C_VEL
LIN {X 0,Y 396.331,Z 912.034,A -85,B 0,C 180,E1 17332.919,E2 17332.919} C_VEL
LIN {X 0,Y 397.996,Z 897.81,A -85,B 0,C 180,E1 17331.612,E2 17331.612} C_VEL
LIN {X 0,Y 399.46,Z 882.485,A -85,B 0,C 180,E1 17330.523,E2 17330.523} C_VEL
LIN {X 0,Y 400.592,Z 865.994,A -85,B 0,C 180,E1 17329.661,E2 17329.661} C_VEL
LIN {X 0,Y 401.316,Z 849.063,A -85,B 0,C 180,E1 17329.058,E2 17329.058} C_VEL
LIN {X 0,Y 403.911,Z 750.25,A -85,B 0,C 180,E1 17327.139,E2 17327.139} C_VEL
LIN {X 0,Y 404.394,Z 725.33,A -85,B 0,C 180,E1 17326.657,E2 17326.657} C_VEL
LIN {X 0,Y 397.786,Z 696.431,A -85,B 0,C 180,E1 17325.37,E2 17325.37} C_VEL
LIN {X 0,Y 398.166,Z 691.929,A -85,B 0,C 180,E1 17324.712,E2 17324.712} C_VEL
LIN {X 0,Y 400.495,Z 673.012,A -85,B 0,C 180,E1 17321.613,E2 17321.613} C_VEL
LIN {X 0,Y 396.992,Z 659.371,A -85,B 0,C 180,E1 17318.654,E2 17318.654} C_VEL
LIN {X 0,Y 393.029,Z 646.656,A -85,B 0,C 180,E1 17315.632,E2 17315.632} C_VEL
LIN {X 0,Y 389.201,Z 635.869,A -85,B 0,C 180,E1 17312.824,E2 17312.824} C_VEL
LIN {X 0,Y 385.635,Z 626.315,A -85,B 0,C 180,E1 17310.07,E2 17310.07} C_VEL
LIN {X 0,Y 385.619,Z 626.189,A -85,B 0,C 180,E1 17305.989,E2 17305.989} C_VEL
LIN {X 0,Y 385.624,Z 626.186,A -85,B 0,C 180,E1 17301.924,E2 17301.924} C_VEL
LIN {X 0,Y 385.619,Z 626.187,A -85,B 0,C 180,E1 17297.816,E2 17297.816} C_VEL
LIN {X 0,Y 385.622,Z 626.184,A -85,B 0,C 180,E1 17293.801,E2 17293.801} C_VEL
LIN {X 0,Y 385.618,Z 626.182,A -85,B 0,C 180,E1 17289.703,E2 17289.703} C_VEL
LIN {X 0,Y 385.618,Z 626.181,A -85,B 0,C 180,E1 17285.804,E2 17285.804} C_VEL
LIN {X 0,Y 385.62,Z 626.188,A -85,B 0,C 180,E1 17281.783,E2 17281.783} C_VEL
LIN {X 0,Y 385.622,Z 626.199,A -85,B 0,C 180,E1 17277.771,E2 17277.771} C_VEL
LIN {X 0,Y 385.622,Z 626.196,A -85,B 0,C 180,E1 17273.748,E2 17273.748} C_VEL
LIN {X 0,Y 385.615,Z 626.187,A -85,B 0,C 180,E1 17269.694,E2 17269.694} C_VEL
LIN {X 0,Y 385.608,Z 626.18,A -85,B 0,C 180,E1 17265.74,E2 17265.74} C_VEL
LIN {X 0,Y 385.605,Z 626.181,A -85,B 0,C 180,E1 17261.715,E2 17261.715} C_VEL
LIN {X 0,Y 385.604,Z 626.189,A -85,B 0,C 180,E1 17257.755,E2 17257.755} C_VEL
LIN {X 0,Y 385.607,Z 626.193,A -85,B 0,C 180,E1 17253.68,E2 17253.68} C_VEL
LIN {X 0,Y 385.612,Z 626.19,A -85,B 0,C 180,E1 17249.628,E2 17249.628} C_VEL
LIN {X 0,Y 385.613,Z 626.189,A -85,B 0,C 180,E1 17245.58,E2 17245.58} C_VEL
LIN {X 0,Y 385.62,Z 626.189,A -85,B 0,C 180,E1 17241.517,E2 17241.517} C_VEL
LIN {X 0,Y 385.628,Z 626.395,A -85,B 0,C 180,E1 17238.809,E2 17238.809} C_VEL
LIN {X 0,Y 387.233,Z 630.135,A -85,B 0,C 180,E1 17237.821,E2 17237.821} C_VEL
LIN {X 0,Y 392.653,Z 642.779,A -85,B 0,C 180,E1 17234.936,E2 17234.936} C_VEL
LIN {X 0,Y 398.561,Z 657.706,A -85,B 0,C 180,E1 17231.942,E2 17231.942} C_VEL
LIN {X 0,Y 403.667,Z 672.829,A -85,B 0,C 180,E1 17229.293,E2 17229.293} C_VEL
LIN {X 0,Y 405.772,Z 680.175,A -85,B 0,C 180,E1 17228.125,E2 17228.125} C_VEL
LIN {X 0,Y 402.145,Z 707.472,A -85,B 0,C 180,E1 17225.19,E2 17225.19} C_VEL
LIN {X 0,Y 406.234,Z 741.164,A -85,B 0,C 180,E1 17224.083,E2 17224.083} C_VEL
LIN {X 0,Y 401.893,Z 915.851,A -85,B 0,C 180,E1 17220.84,E2 17220.84} C_VEL
LIN {X 0,Y 400.663,Z 934.956,A -85,B 0,C 180,E1 17220.245,E2 17220.245} C_VEL
LIN {X 0,Y 399.019,Z 953.3,A -85,B 0,C 180,E1 17219.415,E2 17219.415} C_VEL
LIN {X 0,Y 397.114,Z 971.121,A -85,B 0,C 180,E1 17218.333,E2 17218.333} C_VEL
LIN {X 0,Y 395.054,Z 988.17,A -85,B 0,C 180,E1 17217.015,E2 17217.015} C_VEL
LIN {X 0,Y 392.951,Z 1004.328,A -85,B 0,C 180,E1 17215.468,E2 17215.468} C_VEL
LIN {X 0,Y 390.888,Z 1019.708,A -85,B 0,C 180,E1 17213.677,E2 17213.677} C_VEL
LIN {X 0,Y 388.987,Z 1034.149,A -85,B 0,C 180,E1 17211.645,E2 17211.645} C_VEL
LIN {X 0,Y 387.379,Z 1047.121,A -85,B 0,C 180,E1 17209.448,E2 17209.448} C_VEL
LIN {X 0,Y 386.093,Z 1059.031,A -85,B 0,C 180,E1 17207.015,E2 17207.015} C_VEL
LIN {X 0,Y 385.2,Z 1069.41,A -85,B 0,C 180,E1 17204.429,E2 17204.429} C_VEL
LIN {X 0,Y 384.721,Z 1077.758,A -85,B 0,C 180,E1 17201.848,E2 17201.848} C_VEL
LIN {X 0,Y 384.543,Z 1084.63,A -85,B 0,C 180,E1 17199.126,E2 17199.126} C_VEL
LIN {X 0,Y 384.572,Z 1089.636,A -85,B 0,C 180,E1 17196.419,E2 17196.419} C_VEL
LIN {X 0,Y 384.695,Z 1092.88,A -85,B 0,C 180,E1 17193.725,E2 17193.725} C_VEL
LIN {X 0,Y 384.781,Z 1094.415,A -85,B 0,C 180,E1 17191.042,E2 17191.042} C_VEL
LIN {X 0,Y 384.765,Z 1094.324,A -85,B 0,C 180,E1 17188.511,E2 17188.511} C_VEL
LIN {X 0,Y 384.665,Z 1092.553,A -85,B 0,C 180,E1 17185.826,E2 17185.826} C_VEL
LIN {X 0,Y 384.548,Z 1089.027,A -85,B 0,C 180,E1 17183.13,E2 17183.13} C_VEL
LIN {X 0,Y 384.55,Z 1083.698,A -85,B 0,C 180,E1 17180.421,E2 17180.421} C_VEL
LIN {X 0,Y 384.78,Z 1076.455,A -85,B 0,C 180,E1 17177.697,E2 17177.697} C_VEL
LIN {X 0,Y 385.338,Z 1067.669,A -85,B 0,C 180,E1 17175.114,E2 17175.114} C_VEL
LIN {X 0,Y 386.296,Z 1056.71,A -85,B 0,C 180,E1 17172.527,E2 17172.527} C_VEL
LIN {X 0,Y 387.567,Z 1044.95,A -85,B 0,C 180,E1 17170.247,E2 17170.247} C_VEL
LIN {X 0,Y 389.144,Z 1031.776,A -85,B 0,C 180,E1 17168.126,E2 17168.126} C_VEL
LIN {X 0,Y 390.98,Z 1017.091,A -85,B 0,C 180,E1 17166.168,E2 17166.168} C_VEL
LIN {X 0,Y 392.935,Z 1001.483,A -85,B 0,C 180,E1 17164.449,E2 17164.449} C_VEL
LIN {X 0,Y 394.886,Z 985.029,A -85,B 0,C 180,E1 17162.967,E2 17162.967} C_VEL
LIN {X 0,Y 396.768,Z 967.789,A -85,B 0,C 180,E1 17161.721,E2 17161.721} C_VEL
LIN {X 0,Y 398.465,Z 949.685,A -85,B 0,C 180,E1 17160.704,E2 17160.704} C_VEL
LIN {X 0,Y 399.921,Z 930.935,A -85,B 0,C 180,E1 17159.936,E2 17159.936} C_VEL
LIN {X 0,Y 400.88,Z 911.498,A -85,B 0,C 180,E1 17159.406,E2 17159.406} C_VEL
LIN {X 0,Y 404.362,Z 739.096,A -85,B 0,C 180,E1 17156.294,E2 17156.294} C_VEL
LIN {X 0,Y 400.45,Z 707.089,A -85,B 0,C 180,E1 17155.343,E2 17155.343} C_VEL
LIN {X 0,Y 403.776,Z 677.415,A -85,B 0,C 180,E1 17152.24,E2 17152.24} C_VEL
LIN {X 0,Y 396.182,Z 655.002,A -85,B 0,C 180,E1 17148.88,E2 17148.88} C_VEL
LIN {X 0,Y 389.319,Z 636.157,A -85,B 0,C 180,E1 17145.769,E2 17145.769} C_VEL
LIN {X 0,Y 385.651,Z 626.416,A -85,B 0,C 180,E1 17143.982,E2 17143.982} C_VEL
LIN {X 0,Y 385.623,Z 626.202,A -85,B 0,C 180,E1 17140.017,E2 17140.017} C_VEL
LIN {X 0,Y 385.615,Z 626.202,A -85,B 0,C 180,E1 17136.002,E2 17136.002} C_VEL
LIN {X 0,Y 385.611,Z 626.203,A -85,B 0,C 180,E1 17131.935,E2 17131.935} C_VEL
LIN {X 0,Y 385.607,Z 626.201,A -85,B 0,C 180,E1 17127.846,E2 17127.846} C_VEL
LIN {X 0,Y 385.6,Z 626.205,A -85,B 0,C 180,E1 17123.747,E2 17123.747} C_VEL
LIN {X 0,Y 385.596,Z 626.206,A -85,B 0,C 180,E1 17119.7,E2 17119.7} C_VEL
LIN {X 0,Y 385.649,Z 626.41,A -85,B 0,C 180,E1 17116.725,E2 17116.725} C_VEL
LIN {X 0,Y 386.963,Z 629.76,A -85,B 0,C 180,E1 17116.012,E2 17116.012} C_VEL
LIN {X 0,Y 391.017,Z 638.883,A -85,B 0,C 180,E1 17114.271,E2 17114.271} C_VEL
LIN {X 0,Y 395.723,Z 651.428,A -85,B 0,C 180,E1 17112.088,E2 17112.088} C_VEL
LIN {X 0,Y 399.576,Z 665.214,A -85,B 0,C 180,E1 17109.942,E2 17109.942} C_VEL
LIN {X 0,Y 400.25,Z 669.003,A -85,B 0,C 180,E1 17109.417,E2 17109.417} C_VEL
LIN {X 0,Y 399.113,Z 703.302,A -85,B 0,C 180,E1 17105.246,E2 17105.246} C_VEL
LIN {X 0,Y 398.535,Z 723.505,A -85,B 0,C 180,E1 17102.804,E2 17102.804} C_VEL
LIN {X 0,Y 398.717,Z 727.115,A -85,B 0,C 180,E1 17102.69,E2 17102.69} C_VEL
LIN {X 0,Y 395.03,Z 851.916,A -85,B 0,C 180,E1 17099.927,E2 17099.927} C_VEL
LIN {X 0,Y 394.897,Z 870.062,A -85,B 0,C 180,E1 17099.388,E2 17099.388} C_VEL
LIN {X 0,Y 394.42,Z 886.19,A -85,B 0,C 180,E1 17098.62,E2 17098.62} C_VEL
LIN {X 0,Y 393.719,Z 900.73,A -85,B 0,C 180,E1 17097.669,E2 17097.669} C_VEL
LIN {X 0,Y 392.719,Z 915.253,A -85,B 0,C 180,E1 17096.41,E2 17096.41} C_VEL
LIN {X 0,Y 391.666,Z 927.882,A -85,B 0,C 180,E1 17095.02,E2 17095.02} C_VEL
LIN {X 0,Y 390.478,Z 939.66,A -85,B 0,C 180,E1 17093.383,E2 17093.383} C_VEL
LIN {X 0,Y 389.34,Z 950.051,A -85,B 0,C 180,E1 17091.582,E2 17091.582} C_VEL
LIN {X 0,Y 388.279,Z 958.968,A -85,B 0,C 180,E1 17089.615,E2 17089.615} C_VEL
LIN {X 0,Y 387.376,Z 966.489,A -85,B 0,C 180,E1 17087.478,E2 17087.478} C_VEL
LIN {X 0,Y 386.634,Z 972.399,A -85,B 0,C 180,E1 17085.166,E2 17085.166} C_VEL
LIN {X 0,Y 386.112,Z 976.435,A -85,B 0,C 180,E1 17082.83,E2 17082.83} C_VEL
LIN {X 0,Y 385.77,Z 978.722,A -85,B 0,C 180,E1 17080.309,E2 17080.309} C_VEL
LIN {X 0,Y 385.619,Z 979.051,A -85,B 0,C 180,E1 17077.916,E2 17077.916} C_VEL
LIN {X 0,Y 385.609,Z 977.551,A -85,B 0,C 180,E1 17075.489,E2 17075.489} C_VEL
LIN {X 0,Y 385.751,Z 974.418,A -85,B 0,C 180,E1 17073.191,E2 17073.191} C_VEL
LIN {X 0,Y 386.091,Z 969.214,A -85,B 0,C 180,E1 17070.778,E2 17070.778} C_VEL
LIN {X 0,Y 386.594,Z 962.613,A -85,B 0,C 180,E1 17068.594,E2 17068.594} C_VEL
LIN {X 0,Y 387.29,Z 954.19,A -85,B 0,C 180,E1 17066.462,E2 17066.462} C_VEL
LIN {X 0,Y 388.148,Z 944.234,A -85,B 0,C 180,E1 17064.49,E2 17064.49} C_VEL
LIN {X 0,Y 389.131,Z 932.734,A -85,B 0,C 180,E1 17062.67,E2 17062.67} C_VEL
LIN {X 0,Y 390.109,Z 920.301,A -85,B 0,C 180,E1 17061.101,E2 17061.101} C_VEL
LIN {X 0,Y 391.072,Z 906.395,A -85,B 0,C 180,E1 17059.695,E2 17059.695} C_VEL
LIN {X 0,Y 391.897,Z 891.83,A -85,B 0,C 180,E1 17058.551,E2 17058.551} C_VEL
LIN {X 0,Y 392.584,Z 876.072,A -85,B 0,C 180,E1 17057.612,E2 17057.612} C_VEL
LIN {X 0,Y 392.994,Z 859.265,A -85,B 0,C 180,E1 17056.921,E2 17056.921} C_VEL
LIN {X 0,Y 393.154,Z 839.956,A -85,B 0,C 180,E1 17056.444,E2 17056.444} C_VEL
LIN {X 0,Y 395.664,Z 720.766,A -85,B 0,C 180,E1 17053.991,E2 17053.991} C_VEL
LIN {X 0,Y 394.266,Z 712.924,A -85,B 0,C 180,E1 17053.717,E2 17053.717} C_VEL
LIN {X 0,Y 395.337,Z 682.355,A -85,B 0,C 180,E1 17049.877,E2 17049.877} C_VEL
LIN {X 0,Y 395.854,Z 662.125,A -85,B 0,C 180,E1 17047.316,E2 17047.316} C_VEL
LIN {X 0,Y 390.982,Z 643.759,A -85,B 0,C 180,E1 17044.568,E2 17044.568} C_VEL
LIN {X 0,Y 385.625,Z 626.379,A -85,B 0,C 180,E1 17041.803,E2 17041.803} C_VEL
LIN {X 0,Y 385.581,Z 626.204,A -85,B 0,C 180,E1 17037.993,E2 17037.993} C_VEL
LIN {X 0,Y 385.571,Z 626.165,A -85,B 0,C 180,E1 17034.025,E2 17034.025} C_VEL
LIN {X 0,Y 385.613,Z 626.176,A -85,B 0,C 180,E1 17033.011,E2 17033.011} C_VEL
LIN {X 0,Y 385.383,Z 626.918,A -85,B 0,C 180,E1 17032.368,E2 17032.368} C_VEL
LIN {X 0,Y 384.631,Z 629.932,A -85,B 0,C 180,E1 17031.484,E2 17031.484} C_VEL
LIN {X 0,Y 383.153,Z 637.956,A -85,B 0,C 180,E1 17030.054,E2 17030.054} C_VEL
LIN {X 0,Y 383.004,Z 643.853,A -85,B 0,C 180,E1 17029.008,E2 17029.008} C_VEL
LIN {X 0,Y 383.415,Z 645.866,A -85,B 0,C 180,E1 17028.604,E2 17028.604} C_VEL
LIN {X 0,Y 387.7,Z 661.562,A -85,B 0,C 180,E1 17025.405,E2 17025.405} C_VEL
LIN {X 0,Y 389.767,Z 669.865,A -85,B 0,C 180,E1 17023.803,E2 17023.803} C_VEL
LIN {X 0,Y 387.114,Z 695.343,A -85,B 0,C 180,E1 17019.778,E2 17019.778} C_VEL
LIN {X 0,Y 390.39,Z 712.168,A -85,B 0,C 180,E1 17019.142,E2 17019.142} C_VEL
LIN {X 0,Y 393.062,Z 726.754,A -85,B 0,C 180,E1 17018.653,E2 17018.653} C_VEL
LIN {X 0,Y 390.377,Z 847.888,A -85,B 0,C 180,E1 17016.351,E2 17016.351} C_VEL
LIN {X 0,Y 389.744,Z 865.097,A -85,B 0,C 180,E1 17015.743,E2 17015.743} C_VEL
LIN {X 0,Y 388.764,Z 881.797,A -85,B 0,C 180,E1 17014.869,E2 17014.869} C_VEL
LIN {X 0,Y 387.504,Z 897.114,A -85,B 0,C 180,E1 17013.773,E2 17013.773} C_VEL
LIN {X 0,Y 385.986,Z 912.209,A -85,B 0,C 180,E1 17012.376,E2 17012.376} C_VEL
LIN {X 0,Y 384.467,Z 925.481,A -85,B 0,C 180,E1 17010.82,E2 17010.82} C_VEL
LIN {X 0,Y 382.971,Z 937.226,A -85,B 0,C 180,E1 17009.103,E2 17009.103} C_VEL
LIN {X 0,Y 381.453,Z 948.517,A -85,B 0,C 180,E1 17007.055,E2 17007.055} C_VEL
LIN {X 0,Y 380.152,Z 958.01,A -85,B 0,C 180,E1 17004.87,E2 17004.87} C_VEL
LIN {X 0,Y 379.076,Z 966.221,A -85,B 0,C 180,E1 17002.422,E2 17002.422} C_VEL
LIN {X 0,Y 378.38,Z 972.038,A -85,B 0,C 180,E1 17000.11,E2 17000.11} C_VEL
LIN {X 0,Y 377.913,Z 976.39,A -85,B 0,C 180,E1 16997.626,E2 16997.626} C_VEL
LIN {X 0,Y 377.682,Z 979.182,A -85,B 0,C 180,E1 16994.963,E2 16994.963} C_VEL
LIN {X 0,Y 377.686,Z 980.092,A -85,B 0,C 180,E1 16992.373,E2 16992.373} C_VEL
LIN {X 0,Y 377.923,Z 979.218,A -85,B 0,C 180,E1 16989.722,E2 16989.722} C_VEL
LIN {X 0,Y 378.421,Z 976.641,A -85,B 0,C 180,E1 16987.145,E2 16987.145} C_VEL
LIN {X 0,Y 379.169,Z 972.446,A -85,B 0,C 180,E1 16984.711,E2 16984.711} C_VEL
LIN {X 0,Y 380.271,Z 966.399,A -85,B 0,C 180,E1 16982.265,E2 16982.265} C_VEL
LIN {X 0,Y 381.686,Z 958.865,A -85,B 0,C 180,E1 16979.978,E2 16979.978} C_VEL
LIN {X 0,Y 383.346,Z 949.807,A -85,B 0,C 180,E1 16977.854,E2 16977.854} C_VEL
LIN {X 0,Y 385.27,Z 938.847,A -85,B 0,C 180,E1 16975.816,E2 16975.816} C_VEL
LIN {X 0,Y 387.231,Z 926.829,A -85,B 0,C 180,E1 16974.026,E2 16974.026} C_VEL
LIN {X 0,Y 389.11,Z 913.813,A -85,B 0,C 180,E1 16972.483,E2 16972.483} C_VEL
LIN {X 0,Y 390.929,Z 899.176,A -85,B 0,C 180,E1 16971.105,E2 16971.105} C_VEL
LIN {X 0,Y 392.46,Z 884.208,A -85,B 0,C 180,E1 16970.011,E2 16970.011} C_VEL
LIN {X 0,Y 393.668,Z 867.818,A -85,B 0,C 180,E1 16969.126,E2 16969.126} C_VEL
LIN {X 0,Y 394.459,Z 850.826,A -85,B 0,C 180,E1 16968.496,E2 16968.496} C_VEL
LIN {X 0,Y 395.74,Z 803.152,A -85,B 0,C 180,E1 16967.511,E2 16967.511} C_VEL
LIN {X 0,Y 397.754,Z 726.808,A -85,B 0,C 180,E1 16966.038,E2 16966.038} C_VEL
LIN {X 0,Y 390.855,Z 696.612,A -85,B 0,C 180,E1 16964.643,E2 16964.643} C_VEL
LIN {X 0,Y 391.218,Z 692.521,A -85,B 0,C 180,E1 16964.041,E2 16964.041} C_VEL
LIN {X 0,Y 393.325,Z 675.93,A -85,B 0,C 180,E1 16961.275,E2 16961.275} C_VEL
LIN {X 0,Y 389.792,Z 662.062,A -85,B 0,C 180,E1 16958.185,E2 16958.185} C_VEL
LIN {X 0,Y 385.672,Z 648.886,A -85,B 0,C 180,E1 16954.956,E2 16954.956} C_VEL
LIN {X 0,Y 381.463,Z 637.208,A -85,B 0,C 180,E1 16951.793,E2 16951.793} C_VEL
LIN {X 0,Y 378.517,Z 629.879,A -85,B 0,C 180,E1 16949.602,E2 16949.602} C_VEL
LIN {X 0,Y 377.693,Z 627.28,A -85,B 0,C 180,E1 16948.747,E2 16948.747} C_VEL
LIN {X 0,Y 377.681,Z 627.182,A -85,B 0,C 180,E1 16944.56,E2 16944.56} C_VEL
LIN {X 0,Y 377.682,Z 627.19,A -85,B 0,C 180,E1 16940.42,E2 16940.42} C_VEL
LIN {X 0,Y 377.682,Z 627.191,A -85,B 0,C 180,E1 16936.298,E2 16936.298} C_VEL
LIN {X 0,Y 377.683,Z 627.19,A -85,B 0,C 180,E1 16932.227,E2 16932.227} C_VEL
LIN {X 0,Y 377.683,Z 627.188,A -85,B 0,C 180,E1 16928.066,E2 16928.066} C_VEL
LIN {X 0,Y 377.68,Z 627.184,A -85,B 0,C 180,E1 16923.947,E2 16923.947} C_VEL
LIN {X 0,Y 377.688,Z 627.17,A -85,B 0,C 180,E1 16919.849,E2 16919.849} C_VEL
LIN {X 0,Y 377.678,Z 627.164,A -85,B 0,C 180,E1 16915.749,E2 16915.749} C_VEL
LIN {X 0,Y 377.677,Z 627.171,A -85,B 0,C 180,E1 16911.781,E2 16911.781} C_VEL
LIN {X 0,Y 377.676,Z 627.185,A -85,B 0,C 180,E1 16907.618,E2 16907.618} C_VEL
LIN {X 0,Y 377.675,Z 627.19,A -85,B 0,C 180,E1 16903.545,E2 16903.545} C_VEL
LIN {X 0,Y 377.675,Z 627.19,A -85,B 0,C 180,E1 16899.384,E2 16899.384} C_VEL
LIN {X 0,Y 377.67,Z 627.187,A -85,B 0,C 180,E1 16895.273,E2 16895.273} C_VEL
LIN {X 0,Y 377.668,Z 627.187,A -85,B 0,C 180,E1 16891.195,E2 16891.195} C_VEL
LIN {X 0,Y 377.666,Z 627.194,A -85,B 0,C 180,E1 16887.06,E2 16887.06} C_VEL
LIN {X 0,Y 377.664,Z 627.188,A -85,B 0,C 180,E1 16883.06,E2 16883.06} C_VEL
LIN {X 0,Y 377.718,Z 627.39,A -85,B 0,C 180,E1 16880.119,E2 16880.119} C_VEL
LIN {X 0,Y 379.125,Z 630.896,A -85,B 0,C 180,E1 16879.153,E2 16879.153} C_VEL
LIN {X 0,Y 383.207,Z 639.983,A -85,B 0,C 180,E1 16876.874,E2 16876.874} C_VEL
LIN {X 0,Y 388.743,Z 653.271,A -85,B 0,C 180,E1 16873.932,E2 16873.932} C_VEL
LIN {X 0,Y 394.141,Z 668.058,A -85,B 0,C 180,E1 16871.074,E2 16871.074} C_VEL
LIN {X 0,Y 398.748,Z 682.904,A -85,B 0,C 180,E1 16868.543,E2 16868.543} C_VEL
LIN {X 0,Y 395.331,Z 707.346,A -85,B 0,C 180,E1 16865.868,E2 16865.868} C_VEL
LIN {X 0,Y 399.496,Z 742.005,A -85,B 0,C 180,E1 16864.688,E2 16864.688} C_VEL
LIN {X 0,Y 394.931,Z 915.026,A -85,B 0,C 180,E1 16861.419,E2 16861.419} C_VEL
LIN {X 0,Y 393.647,Z 934.096,A -85,B 0,C 180,E1 16860.816,E2 16860.816} C_VEL
LIN {X 0,Y 391.957,Z 951.987,A -85,B 0,C 180,E1 16859.999,E2 16859.999} C_VEL
LIN {X 0,Y 389.918,Z 970.178,A -85,B 0,C 180,E1 16858.881,E2 16858.881} C_VEL
LIN {X 0,Y 387.78,Z 986.923,A -85,B 0,C 180,E1 16857.569,E2 16857.569} C_VEL
LIN {X 0,Y 385.554,Z 1003.149,A -85,B 0,C 180,E1 16855.993,E2 16855.993} C_VEL
LIN {X 0,Y 383.359,Z 1018.508,A -85,B 0,C 180,E1 16854.172,E2 16854.172} C_VEL
LIN {X 0,Y 381.328,Z 1032.933,A -85,B 0,C 180,E1 16852.102,E2 16852.102} C_VEL
LIN {X 0,Y 379.613,Z 1045.92,A -85,B 0,C 180,E1 16849.863,E2 16849.863} C_VEL
LIN {X 0,Y 378.233,Z 1057.833,A -85,B 0,C 180,E1 16847.38,E2 16847.38} C_VEL
LIN {X 0,Y 377.269,Z 1068.399,A -85,B 0,C 180,E1 16844.683,E2 16844.683} C_VEL
LIN {X 0,Y 376.747,Z 1076.992,A -85,B 0,C 180,E1 16841.947,E2 16841.947} C_VEL
LIN {X 0,Y 376.578,Z 1083.769,A -85,B 0,C 180,E1 16839.166,E2 16839.166} C_VEL
LIN {X 0,Y 376.63,Z 1088.678,A -85,B 0,C 180,E1 16836.401,E2 16836.401} C_VEL
LIN {X 0,Y 376.775,Z 1091.824,A -85,B 0,C 180,E1 16833.651,E2 16833.651} C_VEL
LIN {X 0,Y 376.872,Z 1093.255,A -85,B 0,C 180,E1 16830.912,E2 16830.912} C_VEL
LIN {X 0,Y 376.852,Z 1093.051,A -85,B 0,C 180,E1 16828.327,E2 16828.327} C_VEL
LIN {X 0,Y 376.739,Z 1091.33,A -85,B 0,C 180,E1 16825.738,E2 16825.738} C_VEL
LIN {X 0,Y 376.601,Z 1087.776,A -85,B 0,C 180,E1 16822.985,E2 16822.985} C_VEL
LIN {X 0,Y 376.598,Z 1082.404,A -85,B 0,C 180,E1 16820.216,E2 16820.216} C_VEL
LIN {X 0,Y 376.838,Z 1075.104,A -85,B 0,C 180,E1 16817.433,E2 16817.433} C_VEL
LIN {X 0,Y 377.429,Z 1066.255,A -85,B 0,C 180,E1 16814.795,E2 16814.795} C_VEL
LIN {X 0,Y 378.379,Z 1055.935,A -85,B 0,C 180,E1 16812.308,E2 16812.308} C_VEL
LIN {X 0,Y 379.809,Z 1043.318,A -85,B 0,C 180,E1 16809.826,E2 16809.826} C_VEL
LIN {X 0,Y 381.478,Z 1030.012,A -85,B 0,C 180,E1 16807.663,E2 16807.663} C_VEL
LIN {X 0,Y 383.422,Z 1015.185,A -85,B 0,C 180,E1 16805.668,E2 16805.668} C_VEL
LIN {X 0,Y 385.488,Z 999.412,A -85,B 0,C 180,E1 16803.92,E2 16803.92} C_VEL
LIN {X 0,Y 387.548,Z 982.679,A -85,B 0,C 180,E1 16802.412,E2 16802.412} C_VEL
LIN {X 0,Y 389.524,Z 965.034,A -85,B 0,C 180,E1 16801.146,E2 16801.146} C_VEL
LIN {X 0,Y 391.324,Z 946.311,A -85,B 0,C 180,E1 16800.116,E2 16800.116} C_VEL
LIN {X 0,Y 392.783,Z 927.243,A -85,B 0,C 180,E1 16799.362,E2 16799.362} C_VEL
LIN {X 0,Y 393.662,Z 908.034,A -85,B 0,C 180,E1 16798.866,E2 16798.866} C_VEL
LIN {X 0,Y 397.208,Z 740.049,A -85,B 0,C 180,E1 16795.79,E2 16795.79} C_VEL
LIN {X 0,Y 393.238,Z 706.876,A -85,B 0,C 180,E1 16794.783,E2 16794.783} C_VEL
LIN {X 0,Y 396.407,Z 679.938,A -85,B 0,C 180,E1 16791.902,E2 16791.902} C_VEL
LIN {X 0,Y 388.784,Z 657.3,A -85,B 0,C 180,E1 16788.431,E2 16788.431} C_VEL
LIN {X 0,Y 381.484,Z 637.374,A -85,B 0,C 180,E1 16785.045,E2 16785.045} C_VEL
LIN {X 0,Y 377.702,Z 627.371,A -85,B 0,C 180,E1 16783.141,E2 16783.141} C_VEL
LIN {X 0,Y 377.682,Z 627.182,A -85,B 0,C 180,E1 16779.055,E2 16779.055} C_VEL
LIN {X 0,Y 377.683,Z 627.189,A -85,B 0,C 180,E1 16775.063,E2 16775.063} C_VEL
LIN {X 0,Y 377.687,Z 627.187,A -85,B 0,C 180,E1 16770.902,E2 16770.902} C_VEL
LIN {X 0,Y 377.689,Z 627.19,A -85,B 0,C 180,E1 16766.855,E2 16766.855} C_VEL
LIN {X 0,Y 377.691,Z 627.188,A -85,B 0,C 180,E1 16762.737,E2 16762.737} C_VEL
LIN {X 0,Y 377.688,Z 627.19,A -85,B 0,C 180,E1 16758.604,E2 16758.604} C_VEL
LIN {X 0,Y 377.714,Z 627.549,A -85,B 0,C 180,E1 16757.882,E2 16757.882} C_VEL
LIN {X 0,Y 379.251,Z 631.071,A -85,B 0,C 180,E1 16757.095,E2 16757.095} C_VEL
LIN {X 0,Y 383.755,Z 640.821,A -85,B 0,C 180,E1 16755.102,E2 16755.102} C_VEL
LIN {X 0,Y 388.392,Z 653.064,A -85,B 0,C 180,E1 16752.866,E2 16752.866} C_VEL
LIN {X 0,Y 392.217,Z 666.039,A -85,B 0,C 180,E1 16750.725,E2 16750.725} C_VEL
LIN {X 0,Y 393.429,Z 671.714,A -85,B 0,C 180,E1 16749.877,E2 16749.877} C_VEL
LIN {X 0,Y 392.61,Z 695.156,A -85,B 0,C 180,E1 16747.021,E2 16747.021} C_VEL
LIN {X 0,Y 391.627,Z 725.093,A -85,B 0,C 180,E1 16743.366,E2 16743.366} C_VEL
LIN {X 0,Y 391.791,Z 728.813,A -85,B 0,C 180,E1 16743.25,E2 16743.25} C_VEL
LIN {X 0,Y 387.832,Z 850.548,A -85,B 0,C 180,E1 16740.475,E2 16740.475} C_VEL
LIN {X 0,Y 387.706,Z 869.111,A -85,B 0,C 180,E1 16739.944,E2 16739.944} C_VEL
LIN {X 0,Y 387.305,Z 884.286,A -85,B 0,C 180,E1 16739.26,E2 16739.26} C_VEL
LIN {X 0,Y 386.549,Z 899.464,A -85,B 0,C 180,E1 16738.295,E2 16738.295} C_VEL
LIN {X 0,Y 385.574,Z 913.741,A -85,B 0,C 180,E1 16737.101,E2 16737.101} C_VEL
LIN {X 0,Y 384.364,Z 927.615,A -85,B 0,C 180,E1 16735.599,E2 16735.599} C_VEL
LIN {X 0,Y 383.158,Z 939.285,A -85,B 0,C 180,E1 16734.008,E2 16734.008} C_VEL
LIN {X 0,Y 381.91,Z 949.969,A -85,B 0,C 180,E1 16732.175,E2 16732.175} C_VEL
LIN {X 0,Y 380.749,Z 959.207,A -85,B 0,C 180,E1 16730.172,E2 16730.172} C_VEL
LIN {X 0,Y 379.734,Z 966.928,A -85,B 0,C 180,E1 16727.994,E2 16727.994} C_VEL
LIN {X 0,Y 378.961,Z 972.771,A -85,B 0,C 180,E1 16725.796,E2 16725.796} C_VEL
LIN {X 0,Y 378.346,Z 977.106,A -85,B 0,C 180,E1 16723.416,E2 16723.416} C_VEL
LIN {X 0,Y 377.955,Z 979.643,A -85,B 0,C 180,E1 16721.01,E2 16721.01} C_VEL
LIN {X 0,Y 377.742,Z 980.374,A -85,B 0,C 180,E1 16718.575,E2 16718.575} C_VEL
LIN {X 0,Y 377.689,Z 979.461,A -85,B 0,C 180,E1 16716.272,E2 16716.272} C_VEL
LIN {X 0,Y 377.787,Z 976.599,A -85,B 0,C 180,E1 16713.769,E2 16713.769} C_VEL
LIN {X 0,Y 378.077,Z 972.122,A -85,B 0,C 180,E1 16711.401,E2 16711.401} C_VEL
LIN {X 0,Y 378.58,Z 965.537,A -85,B 0,C 180,E1 16709.001,E2 16709.001} C_VEL
LIN {X 0,Y 379.22,Z 958.01,A -85,B 0,C 180,E1 16706.922,E2 16706.922} C_VEL
LIN {X 0,Y 380.127,Z 947.829,A -85,B 0,C 180,E1 16704.739,E2 16704.739} C_VEL
LIN {X 0,Y 381.102,Z 936.894,A -85,B 0,C 180,E1 16702.884,E2 16702.884} C_VEL
LIN {X 0,Y 382.212,Z 923.793,A -85,B 0,C 180,E1 16701.109,E2 16701.109} C_VEL
LIN {X 0,Y 383.224,Z 909.9,A -85,B 0,C 180,E1 16699.628,E2 16699.628} C_VEL
LIN {X 0,Y 384.129,Z 895.467,A -85,B 0,C 180,E1 16698.413,E2 16698.413} C_VEL
LIN {X 0,Y 384.891,Z 879.137,A -85,B 0,C 180,E1 16697.385,E2 16697.385} C_VEL
LIN {X 0,Y 385.361,Z 862.965,A -85,B 0,C 180,E1 16696.661,E2 16696.661} C_VEL
LIN {X 0,Y 385.554,Z 844.403,A -85,B 0,C 180,E1 16696.154,E2 16696.154} C_VEL
LIN {X 0,Y 388.217,Z 721.9,A -85,B 0,C 180,E1 16693.58,E2 16693.58} C_VEL
LIN {X 0,Y 386.822,Z 713.89,A -85,B 0,C 180,E1 16693.285,E2 16693.285} C_VEL
LIN {X 0,Y 387.961,Z 682.717,A -85,B 0,C 180,E1 16689.346,E2 16689.346} C_VEL
LIN {X 0,Y 388.427,Z 664.602,A -85,B 0,C 180,E1 16687.039,E2 16687.039} C_VEL
LIN {X 0,Y 383.591,Z 646.335,A -85,B 0,C 180,E1 16684.265,E2 16684.265} C_VEL
LIN {X 0,Y 377.686,Z 627.382,A -85,B 0,C 180,E1 16681.22,E2 16681.22} C_VEL
LIN {X 0,Y 377.678,Z 627.191,A -85,B 0,C 180,E1 16677.429,E2 16677.429} C_VEL
LIN {X 0,Y 377.68,Z 627.158,A -85,B 0,C 180,E1 16673.233,E2 16673.233} C_VEL
LIN {X 0,Y 377.693,Z 627.492,A -85,B 0,C 180,E1 16672.655,E2 16672.655} C_VEL
LIN {X 0,Y 382.553,Z 642.891,A -85,B 0,C 180,E1 16669.228,E2 16669.228} C_VEL
LIN {X 0,Y 383.415,Z 645.866,A -85,B 0,C 180,E1 16668.604,E2 16668.604} C_VEL
LIN {X 0,Y 383.805,Z 650.754,A -85,B 0,C 180,E1 16667.703,E2 16667.703} C_VEL
LIN {X 0,Y 381.335,Z 665.934,A -85,B 0,C 180,E1 16665.262,E2 16665.262} C_VEL
LIN {X 0,Y 381.647,Z 669.462,A -85,B 0,C 180,E1 16664.613,E2 16664.613} C_VEL
LIN {X 0,Y 382.189,Z 673.119,A -85,B 0,C 180,E1 16663.927,E2 16663.927} C_VEL
LIN {X 0,Y 379.775,Z 695.525,A -85,B 0,C 180,E1 16660.352,E2 16660.352} C_VEL
LIN {X 0,Y 385.902,Z 727.928,A -85,B 0,C 180,E1 16659.166,E2 16659.166} C_VEL
LIN {X 0,Y 383.092,Z 848.679,A -85,B 0,C 180,E1 16656.83,E2 16656.83} C_VEL
LIN {X 0,Y 382.425,Z 865.976,A -85,B 0,C 180,E1 16656.206,E2 16656.206} C_VEL
LIN {X 0,Y 381.428,Z 882.284,A -85,B 0,C 180,E1 16655.34,E2 16655.34} C_VEL
LIN {X 0,Y 380.115,Z 897.722,A -85,B 0,C 180,E1 16654.224,E2 16654.224} C_VEL
LIN {X 0,Y 378.527,Z 912.887,A -85,B 0,C 180,E1 16652.801,E2 16652.801} C_VEL
LIN {X 0,Y 376.937,Z 926.24,A -85,B 0,C 180,E1 16651.216,E2 16651.216} C_VEL
LIN {X 0,Y 375.303,Z 938.497,A -85,B 0,C 180,E1 16649.39,E2 16649.39} C_VEL
LIN {X 0,Y 373.78,Z 949.299,A -85,B 0,C 180,E1 16647.394,E2 16647.394} C_VEL
LIN {X 0,Y 372.445,Z 958.651,A -85,B 0,C 180,E1 16645.227,E2 16645.227} C_VEL
LIN {X 0,Y 371.344,Z 966.506,A -85,B 0,C 180,E1 16642.886,E2 16642.886} C_VEL
LIN {X 0,Y 370.535,Z 972.888,A -85,B 0,C 180,E1 16640.369,E2 16640.369} C_VEL
LIN {X 0,Y 370.03,Z 977.364,A -85,B 0,C 180,E1 16637.833,E2 16637.833} C_VEL
LIN {X 0,Y 369.773,Z 980.249,A -85,B 0,C 180,E1 16635.116,E2 16635.116} C_VEL
LIN {X 0,Y 369.772,Z 981.297,A -85,B 0,C 180,E1 16632.534,E2 16632.534} C_VEL
LIN {X 0,Y 369.993,Z 980.638,A -85,B 0,C 180,E1 16629.928,E2 16629.928} C_VEL
LIN {X 0,Y 370.535,Z 978.073,A -85,B 0,C 180,E1 16627.135,E2 16627.135} C_VEL
LIN {X 0,Y 371.328,Z 974.069,A -85,B 0,C 180,E1 16624.651,E2 16624.651} C_VEL
LIN {X 0,Y 372.478,Z 968.171,A -85,B 0,C 180,E1 16622.156,E2 16622.156} C_VEL
LIN {X 0,Y 374.042,Z 960.379,A -85,B 0,C 180,E1 16619.703,E2 16619.703} C_VEL
LIN {X 0,Y 375.84,Z 951.232,A -85,B 0,C 180,E1 16617.494,E2 16617.494} C_VEL
LIN {X 0,Y 377.923,Z 940.046,A -85,B 0,C 180,E1 16615.367,E2 16615.367} C_VEL
LIN {X 0,Y 380.036,Z 927.846,A -85,B 0,C 180,E1 16613.517,E2 16613.517} C_VEL
LIN {X 0,Y 382.015,Z 914.928,A -85,B 0,C 180,E1 16611.958,E2 16611.958} C_VEL
LIN {X 0,Y 383.945,Z 900.253,A -85,B 0,C 180,E1 16610.549,E2 16610.549} C_VEL
LIN {X 0,Y 385.538,Z 885.58,A -85,B 0,C 180,E1 16609.453,E2 16609.453} C_VEL
LIN {X 0,Y 386.818,Z 869.35,A -85,B 0,C 180,E1 16608.553,E2 16608.553} C_VEL
LIN {X 0,Y 387.674,Z 852.165,A -85,B 0,C 180,E1 16607.896,E2 16607.896} C_VEL
LIN {X 0,Y 388.595,Z 818.872,A -85,B 0,C 180,E1 16607.176,E2 16607.176} C_VEL
LIN {X 0,Y 391.181,Z 728.36,A -85,B 0,C 180,E1 16605.399,E2 16605.399} C_VEL
LIN {X 0,Y 384.376,Z 698.453,A -85,B 0,C 180,E1 16603.978,E2 16603.978} C_VEL
LIN {X 0,Y 383.978,Z 695.847,A -85,B 0,C 180,E1 16603.785,E2 16603.785} C_VEL
LIN {X 0,Y 386.26,Z 679.26,A -85,B 0,C 180,E1 16601.011,E2 16601.011} C_VEL
LIN {X 0,Y 382.873,Z 665.757,A -85,B 0,C 180,E1 16597.94,E2 16597.94} C_VEL
LIN {X 0,Y 378.948,Z 653,A -85,B 0,C 180,E1 16594.745,E2 16594.745} C_VEL
LIN {X 0,Y 374.817,Z 641.423,A -85,B 0,C 180,E1 16591.524,E2 16591.524} C_VEL
LIN {X 0,Y 371.056,Z 631.68,A -85,B 0,C 180,E1 16588.545,E2 16588.545} C_VEL
LIN {X 0,Y 369.758,Z 628.284,A -85,B 0,C 180,E1 16587.368,E2 16587.368} C_VEL
LIN {X 0,Y 369.745,Z 628.17,A -85,B 0,C 180,E1 16583.159,E2 16583.159} C_VEL
LIN {X 0,Y 369.739,Z 628.164,A -85,B 0,C 180,E1 16579.1,E2 16579.1} C_VEL
LIN {X 0,Y 369.734,Z 628.162,A -85,B 0,C 180,E1 16575.047,E2 16575.047} C_VEL
LIN {X 0,Y 369.734,Z 628.163,A -85,B 0,C 180,E1 16570.912,E2 16570.912} C_VEL
LIN {X 0,Y 369.731,Z 628.171,A -85,B 0,C 180,E1 16566.834,E2 16566.834} C_VEL
LIN {X 0,Y 369.733,Z 628.178,A -85,B 0,C 180,E1 16562.635,E2 16562.635} C_VEL
LIN {X 0,Y 369.733,Z 628.18,A -85,B 0,C 180,E1 16558.451,E2 16558.451} C_VEL
LIN {X 0,Y 369.731,Z 628.167,A -85,B 0,C 180,E1 16554.258,E2 16554.258} C_VEL
LIN {X 0,Y 369.728,Z 628.157,A -85,B 0,C 180,E1 16550.191,E2 16550.191} C_VEL
LIN {X 0,Y 369.729,Z 628.156,A -85,B 0,C 180,E1 16546.073,E2 16546.073} C_VEL
LIN {X 0,Y 369.731,Z 628.16,A -85,B 0,C 180,E1 16542.044,E2 16542.044} C_VEL
LIN {X 0,Y 369.733,Z 628.167,A -85,B 0,C 180,E1 16537.921,E2 16537.921} C_VEL
LIN {X 0,Y 369.735,Z 628.171,A -85,B 0,C 180,E1 16533.846,E2 16533.846} C_VEL
LIN {X 0,Y 369.743,Z 628.169,A -85,B 0,C 180,E1 16529.803,E2 16529.803} C_VEL
LIN {X 0,Y 369.74,Z 628.166,A -85,B 0,C 180,E1 16525.773,E2 16525.773} C_VEL
LIN {X 0,Y 369.771,Z 628.355,A -85,B 0,C 180,E1 16521.56,E2 16521.56} C_VEL
LIN {X 0,Y 371.158,Z 631.843,A -85,B 0,C 180,E1 16520.524,E2 16520.524} C_VEL
LIN {X 0,Y 375.494,Z 641.332,A -85,B 0,C 180,E1 16517.98,E2 16517.98} C_VEL
LIN {X 0,Y 380.5,Z 653.172,A -85,B 0,C 180,E1 16515.193,E2 16515.193} C_VEL
LIN {X 0,Y 385.69,Z 666.785,A -85,B 0,C 180,E1 16512.368,E2 16512.368} C_VEL
LIN {X 0,Y 390.445,Z 681.467,A -85,B 0,C 180,E1 16509.689,E2 16509.689} C_VEL
LIN {X 0,Y 391.634,Z 686.241,A -85,B 0,C 180,E1 16508.906,E2 16508.906} C_VEL
LIN {X 0,Y 388.576,Z 706.812,A -85,B 0,C 180,E1 16506.6,E2 16506.6} C_VEL
LIN {X 0,Y 392.32,Z 738.623,A -85,B 0,C 180,E1 16505.461,E2 16505.461} C_VEL
LIN {X 0,Y 392.749,Z 745.192,A -85,B 0,C 180,E1 16505.272,E2 16505.272} C_VEL
LIN {X 0,Y 388.035,Z 914.159,A -85,B 0,C 180,E1 16502.026,E2 16502.026} C_VEL
LIN {X 0,Y 386.694,Z 933.308,A -85,B 0,C 180,E1 16501.412,E2 16501.412} C_VEL
LIN {X 0,Y 384.953,Z 950.847,A -85,B 0,C 180,E1 16500.602,E2 16500.602} C_VEL
LIN {X 0,Y 382.843,Z 968.741,A -85,B 0,C 180,E1 16499.491,E2 16499.491} C_VEL
LIN {X 0,Y 380.545,Z 985.765,A -85,B 0,C 180,E1 16498.139,E2 16498.139} C_VEL
LIN {X 0,Y 378.191,Z 1001.981,A -85,B 0,C 180,E1 16496.538,E2 16496.538} C_VEL
LIN {X 0,Y 375.861,Z 1017.355,A -85,B 0,C 180,E1 16494.686,E2 16494.686} C_VEL
LIN {X 0,Y 373.759,Z 1031.383,A -85,B 0,C 180,E1 16492.643,E2 16492.643} C_VEL
LIN {X 0,Y 371.871,Z 1044.746,A -85,B 0,C 180,E1 16490.294,E2 16490.294} C_VEL
LIN {X 0,Y 370.387,Z 1056.644,A -85,B 0,C 180,E1 16487.76,E2 16487.76} C_VEL
LIN {X 0,Y 369.372,Z 1067.024,A -85,B 0,C 180,E1 16485.062,E2 16485.062} C_VEL
LIN {X 0,Y 368.791,Z 1075.811,A -85,B 0,C 180,E1 16482.208,E2 16482.208} C_VEL
LIN {X 0,Y 368.616,Z 1082.585,A -85,B 0,C 180,E1 16479.366,E2 16479.366} C_VEL
LIN {X 0,Y 368.68,Z 1087.496,A -85,B 0,C 180,E1 16476.54,E2 16476.54} C_VEL
LIN {X 0,Y 368.846,Z 1090.643,A -85,B 0,C 180,E1 16473.73,E2 16473.73} C_VEL
LIN {X 0,Y 368.959,Z 1092.067,A -85,B 0,C 180,E1 16470.931,E2 16470.931} C_VEL
LIN {X 0,Y 368.939,Z 1091.846,A -85,B 0,C 180,E1 16468.291,E2 16468.291} C_VEL
LIN {X 0,Y 368.813,Z 1090.099,A -85,B 0,C 180,E1 16465.646,E2 16465.646} C_VEL
LIN {X 0,Y 368.653,Z 1086.515,A -85,B 0,C 180,E1 16462.833,E2 16462.833} C_VEL
LIN {X 0,Y 368.645,Z 1081.101,A -85,B 0,C 180,E1 16460.003,E2 16460.003} C_VEL
LIN {X 0,Y 368.898,Z 1073.725,A -85,B 0,C 180,E1 16457.158,E2 16457.158} C_VEL
LIN {X 0,Y 369.551,Z 1064.576,A -85,B 0,C 180,E1 16454.407,E2 16454.407} C_VEL
LIN {X 0,Y 370.548,Z 1054.382,A -85,B 0,C 180,E1 16451.922,E2 16451.922} C_VEL
LIN {X 0,Y 371.961,Z 1042.562,A -85,B 0,C 180,E1 16449.546,E2 16449.546} C_VEL
LIN {X 0,Y 373.699,Z 1029.313,A -85,B 0,C 180,E1 16447.338,E2 16447.338} C_VEL
LIN {X 0,Y 375.721,Z 1014.517,A -85,B 0,C 180,E1 16445.303,E2 16445.303} C_VEL
LIN {X 0,Y 377.873,Z 998.762,A -85,B 0,C 180,E1 16443.522,E2 16443.522} C_VEL
LIN {X 0,Y 380.017,Z 982.089,A -85,B 0,C 180,E1 16441.988,E2 16441.988} C_VEL
LIN {X 0,Y 382.068,Z 964.529,A -85,B 0,C 180,E1 16440.7,E2 16440.7} C_VEL
LIN {X 0,Y 383.939,Z 945.924,A -85,B 0,C 180,E1 16439.654,E2 16439.654} C_VEL
LIN {X 0,Y 385.467,Z 926.767,A -85,B 0,C 180,E1 16438.878,E2 16438.878} C_VEL
LIN {X 0,Y 386.385,Z 907.57,A -85,B 0,C 180,E1 16438.371,E2 16438.371} C_VEL
LIN {X 0,Y 390.071,Z 741.036,A -85,B 0,C 180,E1 16435.274,E2 16435.274} C_VEL
LIN {X 0,Y 386.044,Z 706.79,A -85,B 0,C 180,E1 16434.218,E2 16434.218} C_VEL
LIN {X 0,Y 389.107,Z 682.726,A -85,B 0,C 180,E1 16431.604,E2 16431.604} C_VEL
LIN {X 0,Y 381.732,Z 660.755,A -85,B 0,C 180,E1 16428.174,E2 16428.174} C_VEL
LIN {X 0,Y 374.681,Z 641.227,A -85,B 0,C 180,E1 16424.778,E2 16424.778} C_VEL
LIN {X 0,Y 369.768,Z 628.36,A -85,B 0,C 180,E1 16422.271,E2 16422.271} C_VEL
LIN {X 0,Y 369.739,Z 628.174,A -85,B 0,C 180,E1 16418.1,E2 16418.1} C_VEL
LIN {X 0,Y 369.736,Z 628.18,A -85,B 0,C 180,E1 16414.04,E2 16414.04} C_VEL
LIN {X 0,Y 369.731,Z 628.18,A -85,B 0,C 180,E1 16410.019,E2 16410.019} C_VEL
LIN {X 0,Y 369.729,Z 628.179,A -85,B 0,C 180,E1 16405.982,E2 16405.982} C_VEL
LIN {X 0,Y 369.725,Z 628.181,A -85,B 0,C 180,E1 16401.913,E2 16401.913} C_VEL
LIN {X 0,Y 369.756,Z 628.426,A -85,B 0,C 180,E1 16399.31,E2 16399.31} C_VEL
LIN {X 0,Y 371.104,Z 631.739,A -85,B 0,C 180,E1 16398.487,E2 16398.487} C_VEL
LIN {X 0,Y 372.241,Z 633.726,A -85,B 0,C 180,E1 16397.992,E2 16397.992} C_VEL
LIN {X 0,Y 376.099,Z 641.873,A -85,B 0,C 180,E1 16396.209,E2 16396.209} C_VEL
LIN {X 0,Y 380.837,Z 653.595,A -85,B 0,C 180,E1 16393.9,E2 16393.9} C_VEL
LIN {X 0,Y 384.866,Z 666.623,A -85,B 0,C 180,E1 16391.641,E2 16391.641} C_VEL
LIN {X 0,Y 386.66,Z 675.178,A -85,B 0,C 180,E1 16390.278,E2 16390.278} C_VEL
LIN {X 0,Y 385.763,Z 700.242,A -85,B 0,C 180,E1 16387.221,E2 16387.221} C_VEL
LIN {X 0,Y 384.772,Z 726.566,A -85,B 0,C 180,E1 16383.967,E2 16383.967} C_VEL
LIN {X 0,Y 384.965,Z 729.91,A -85,B 0,C 180,E1 16383.853,E2 16383.853} C_VEL
LIN {X 0,Y 380.684,Z 852.294,A -85,B 0,C 180,E1 16380.978,E2 16380.978} C_VEL
LIN {X 0,Y 380.514,Z 870.988,A -85,B 0,C 180,E1 16380.418,E2 16380.418} C_VEL
LIN {X 0,Y 380.055,Z 886.357,A -85,B 0,C 180,E1 16379.698,E2 16379.698} C_VEL
LIN {X 0,Y 379.197,Z 902.386,A -85,B 0,C 180,E1 16378.64,E2 16378.64} C_VEL
LIN {X 0,Y 378.151,Z 916.281,A -85,B 0,C 180,E1 16377.423,E2 16377.423} C_VEL
LIN {X 0,Y 376.875,Z 929.926,A -85,B 0,C 180,E1 16375.892,E2 16375.892} C_VEL
LIN {X 0,Y 375.526,Z 941.831,A -85,B 0,C 180,E1 16374.193,E2 16374.193} C_VEL
LIN {X 0,Y 374.219,Z 952.315,A -85,B 0,C 180,E1 16372.322,E2 16372.322} C_VEL
LIN {X 0,Y 372.994,Z 961.312,A -85,B 0,C 180,E1 16370.277,E2 16370.277} C_VEL
LIN {X 0,Y 371.935,Z 968.884,A -85,B 0,C 180,E1 16368.053,E2 16368.053} C_VEL
LIN {X 0,Y 371.107,Z 974.503,A -85,B 0,C 180,E1 16365.807,E2 16365.807} C_VEL
LIN {X 0,Y 370.461,Z 978.704,A -85,B 0,C 180,E1 16363.363,E2 16363.363} C_VEL
LIN {X 0,Y 370.049,Z 981.027,A -85,B 0,C 180,E1 16360.917,E2 16360.917} C_VEL
LIN {X 0,Y 369.833,Z 981.611,A -85,B 0,C 180,E1 16358.427,E2 16358.427} C_VEL
LIN {X 0,Y 369.779,Z 980.479,A -85,B 0,C 180,E1 16356.056,E2 16356.056} C_VEL
LIN {X 0,Y 369.901,Z 977.394,A -85,B 0,C 180,E1 16353.472,E2 16353.472} C_VEL
LIN {X 0,Y 370.22,Z 972.624,A -85,B 0,C 180,E1 16351.05,E2 16351.05} C_VEL
LIN {X 0,Y 370.771,Z 965.919,A -85,B 0,C 180,E1 16348.636,E2 16348.636} C_VEL
LIN {X 0,Y 371.526,Z 957.327,A -85,B 0,C 180,E1 16346.331,E2 16346.331} C_VEL
LIN {X 0,Y 372.442,Z 947.596,A -85,B 0,C 180,E1 16344.282,E2 16344.282} C_VEL
LIN {X 0,Y 373.564,Z 935.39,A -85,B 0,C 180,E1 16342.257,E2 16342.257} C_VEL
LIN {X 0,Y 374.601,Z 923.33,A -85,B 0,C 180,E1 16340.66,E2 16340.66} C_VEL
LIN {X 0,Y 375.707,Z 908.585,A -85,B 0,C 180,E1 16339.105,E2 16339.105} C_VEL
LIN {X 0,Y 376.647,Z 893.182,A -85,B 0,C 180,E1 16337.858,E2 16337.858} C_VEL
LIN {X 0,Y 377.347,Z 878.273,A -85,B 0,C 180,E1 16336.943,E2 16336.943} C_VEL
LIN {X 0,Y 377.802,Z 861.375,A -85,B 0,C 180,E1 16336.218,E2 16336.218} C_VEL
LIN {X 0,Y 377.994,Z 841.606,A -85,B 0,C 180,E1 16335.707,E2 16335.707} C_VEL
LIN {X 0,Y 380.79,Z 723.037,A -85,B 0,C 180,E1 16333.152,E2 16333.152} C_VEL
LIN {X 0,Y 379.387,Z 714.82,A -85,B 0,C 180,E1 16332.84,E2 16332.84} C_VEL
LIN {X 0,Y 380.574,Z 683.819,A -85,B 0,C 180,E1 16328.897,E2 16328.897} C_VEL
LIN {X 0,Y 381.003,Z 667.064,A -85,B 0,C 180,E1 16326.751,E2 16326.751} C_VEL
LIN {X 0,Y 376.435,Z 649.71,A -85,B 0,C 180,E1 16324.087,E2 16324.087} C_VEL
LIN {X 0,Y 370.608,Z 631.081,A -85,B 0,C 180,E1 16321.108,E2 16321.108} C_VEL
LIN {X 0,Y 369.72,Z 628.383,A -85,B 0,C 180,E1 16320.612,E2 16320.612} C_VEL
LIN {X 0,Y 369.707,Z 628.17,A -85,B 0,C 180,E1 16316.813,E2 16316.813} C_VEL
LIN {X 0,Y 369.737,Z 628.277,A -85,B 0,C 180,E1 16313.545,E2 16313.545} C_VEL
LIN {X 0,Y 372.409,Z 636.465,A -85,B 0,C 180,E1 16311.582,E2 16311.582} C_VEL
LIN {X 0,Y 377.015,Z 651.758,A -85,B 0,C 180,E1 16308.237,E2 16308.237} C_VEL
LIN {X 0,Y 381.315,Z 668.058,A -85,B 0,C 180,E1 16304.891,E2 16304.891} C_VEL
LIN {X 0,Y 381.647,Z 669.462,A -85,B 0,C 180,E1 16304.613,E2 16304.613} C_VEL
LIN {X 0,Y 381.621,Z 673.107,A -85,B 0,C 180,E1 16303.985,E2 16303.985} C_VEL
LIN {X 0,Y 379.658,Z 678.703,A -85,B 0,C 180,E1 16303.204,E2 16303.204} C_VEL
LIN {X 0,Y 373.478,Z 690.969,A -85,B 0,C 180,E1 16301.636,E2 16301.636} C_VEL
LIN {X 0,Y 372.504,Z 694.839,A -85,B 0,C 180,E1 16301.058,E2 16301.058} C_VEL
LIN {X 0,Y 372.678,Z 697.168,A -85,B 0,C 180,E1 16300.866,E2 16300.866} C_VEL
LIN {X 0,Y 378.771,Z 729.197,A -85,B 0,C 180,E1 16299.696,E2 16299.696} C_VEL
LIN {X 0,Y 375.84,Z 849.31,A -85,B 0,C 180,E1 16297.332,E2 16297.332} C_VEL
LIN {X 0,Y 375.149,Z 866.546,A -85,B 0,C 180,E1 16296.701,E2 16296.701} C_VEL
LIN {X 0,Y 374.117,Z 882.759,A -85,B 0,C 180,E1 16295.829,E2 16295.829} C_VEL
LIN {X 0,Y 372.75,Z 898.313,A -85,B 0,C 180,E1 16294.693,E2 16294.693} C_VEL
LIN {X 0,Y 371.087,Z 913.542,A -85,B 0,C 180,E1 16293.244,E2 16293.244} C_VEL
LIN {X 0,Y 369.422,Z 926.97,A -85,B 0,C 180,E1 16291.629,E2 16291.629} C_VEL
LIN {X 0,Y 367.776,Z 938.824,A -85,B 0,C 180,E1 16289.845,E2 16289.845} C_VEL
LIN {X 0,Y 366.161,Z 949.752,A -85,B 0,C 180,E1 16287.81,E2 16287.81} C_VEL
LIN {X 0,Y 364.745,Z 959.259,A -85,B 0,C 180,E1 16285.598,E2 16285.598} C_VEL
LIN {X 0,Y 363.544,Z 967.383,A -85,B 0,C 180,E1 16283.154,E2 16283.154} C_VEL
LIN {X 0,Y 362.695,Z 973.708,A -85,B 0,C 180,E1 16280.64,E2 16280.64} C_VEL
LIN {X 0,Y 362.152,Z 978.328,A -85,B 0,C 180,E1 16278.05,E2 16278.05} C_VEL
LIN {X 0,Y 361.866,Z 981.321,A -85,B 0,C 180,E1 16275.258,E2 16275.258} C_VEL
LIN {X 0,Y 361.864,Z 982.495,A -85,B 0,C 180,E1 16272.472,E2 16272.472} C_VEL
LIN {X 0,Y 362.108,Z 981.854,A -85,B 0,C 180,E1 16269.809,E2 16269.809} C_VEL
LIN {X 0,Y 362.695,Z 979.312,A -85,B 0,C 180,E1 16266.955,E2 16266.955} C_VEL
LIN {X 0,Y 363.547,Z 975.341,A -85,B 0,C 180,E1 16264.419,E2 16264.419} C_VEL
LIN {X 0,Y 364.78,Z 969.481,A -85,B 0,C 180,E1 16261.872,E2 16261.872} C_VEL
LIN {X 0,Y 366.48,Z 961.574,A -85,B 0,C 180,E1 16259.324,E2 16259.324} C_VEL
LIN {X 0,Y 368.351,Z 952.685,A -85,B 0,C 180,E1 16257.12,E2 16257.12} C_VEL
LIN {X 0,Y 370.48,Z 941.95,A -85,B 0,C 180,E1 16255.018,E2 16255.018} C_VEL
LIN {X 0,Y 372.666,Z 930.091,A -85,B 0,C 180,E1 16253.156,E2 16253.156} C_VEL
LIN {X 0,Y 374.755,Z 917.473,A -85,B 0,C 180,E1 16251.564,E2 16251.564} C_VEL
LIN {X 0,Y 376.754,Z 903.251,A -85,B 0,C 180,E1 16250.141,E2 16250.141} C_VEL
LIN {X 0,Y 378.502,Z 888.311,A -85,B 0,C 180,E1 16248.971,E2 16248.971} C_VEL
LIN {X 0,Y 379.891,Z 872.739,A -85,B 0,C 180,E1 16248.048,E2 16248.048} C_VEL
LIN {X 0,Y 380.837,Z 855.884,A -85,B 0,C 180,E1 16247.351,E2 16247.351} C_VEL
LIN {X 0,Y 381.469,Z 834.211,A -85,B 0,C 180,E1 16246.818,E2 16246.818} C_VEL
LIN {X 0,Y 384.657,Z 729.842,A -85,B 0,C 180,E1 16244.731,E2 16244.731} C_VEL
LIN {X 0,Y 377.929,Z 699.998,A -85,B 0,C 180,E1 16243.266,E2 16243.266} C_VEL
LIN {X 0,Y 377.175,Z 696.472,A -85,B 0,C 180,E1 16243.048,E2 16243.048} C_VEL
LIN {X 0,Y 379.126,Z 682.207,A -85,B 0,C 180,E1 16240.648,E2 16240.648} C_VEL
LIN {X 0,Y 375.813,Z 668.887,A -85,B 0,C 180,E1 16237.536,E2 16237.536} C_VEL
LIN {X 0,Y 371.876,Z 655.931,A -85,B 0,C 180,E1 16234.19,E2 16234.19} C_VEL
LIN {X 0,Y 367.645,Z 643.933,A -85,B 0,C 180,E1 16230.75,E2 16230.75} C_VEL
LIN {X 0,Y 364.134,Z 635.398,A -85,B 0,C 180,E1 16228.005,E2 16228.005} C_VEL
LIN {X 0,Y 361.817,Z 629.276,A -85,B 0,C 180,E1 16225.841,E2 16225.841} C_VEL
LIN {X 0,Y 361.799,Z 629.154,A -85,B 0,C 180,E1 16221.565,E2 16221.565} C_VEL
LIN {X 0,Y 361.798,Z 629.157,A -85,B 0,C 180,E1 16217.366,E2 16217.366} C_VEL
LIN {X 0,Y 361.796,Z 629.159,A -85,B 0,C 180,E1 16213.098,E2 16213.098} C_VEL
LIN {X 0,Y 361.796,Z 629.155,A -85,B 0,C 180,E1 16208.903,E2 16208.903} C_VEL
LIN {X 0,Y 361.793,Z 629.149,A -85,B 0,C 180,E1 16204.756,E2 16204.756} C_VEL
LIN {X 0,Y 361.791,Z 629.144,A -85,B 0,C 180,E1 16200.634,E2 16200.634} C_VEL
LIN {X 0,Y 361.789,Z 629.146,A -85,B 0,C 180,E1 16196.515,E2 16196.515} C_VEL
LIN {X 0,Y 361.793,Z 629.158,A -85,B 0,C 180,E1 16192.377,E2 16192.377} C_VEL
LIN {X 0,Y 361.794,Z 629.166,A -85,B 0,C 180,E1 16188.2,E2 16188.2} C_VEL
LIN {X 0,Y 361.792,Z 629.169,A -85,B 0,C 180,E1 16183.957,E2 16183.957} C_VEL
LIN {X 0,Y 361.792,Z 629.16,A -85,B 0,C 180,E1 16179.791,E2 16179.791} C_VEL
LIN {X 0,Y 361.79,Z 629.156,A -85,B 0,C 180,E1 16175.683,E2 16175.683} C_VEL
LIN {X 0,Y 361.791,Z 629.159,A -85,B 0,C 180,E1 16171.438,E2 16171.438} C_VEL
LIN {X 0,Y 361.789,Z 629.167,A -85,B 0,C 180,E1 16167.202,E2 16167.202} C_VEL
LIN {X 0,Y 361.814,Z 629.365,A -85,B 0,C 180,E1 16163.112,E2 16163.112} C_VEL
LIN {X 0,Y 363.507,Z 633.193,A -85,B 0,C 180,E1 16161.875,E2 16161.875} C_VEL
LIN {X 0,Y 367.669,Z 642.346,A -85,B 0,C 180,E1 16159.257,E2 16159.257} C_VEL
LIN {X 0,Y 372.824,Z 654.467,A -85,B 0,C 180,E1 16156.218,E2 16156.218} C_VEL
LIN {X 0,Y 378.135,Z 668.137,A -85,B 0,C 180,E1 16153.223,E2 16153.223} C_VEL
LIN {X 0,Y 382.956,Z 682.678,A -85,B 0,C 180,E1 16150.441,E2 16150.441} C_VEL
LIN {X 0,Y 384.663,Z 688.907,A -85,B 0,C 180,E1 16149.363,E2 16149.363} C_VEL
LIN {X 0,Y 381.875,Z 706.676,A -85,B 0,C 180,E1 16147.332,E2 16147.332} C_VEL
LIN {X 0,Y 385.662,Z 739.142,A -85,B 0,C 180,E1 16146.131,E2 16146.131} C_VEL
LIN {X 0,Y 386.125,Z 746.224,A -85,B 0,C 180,E1 16145.921,E2 16145.921} C_VEL
LIN {X 0,Y 381.193,Z 913.327,A -85,B 0,C 180,E1 16142.657,E2 16142.657} C_VEL
LIN {X 0,Y 379.8,Z 932.373,A -85,B 0,C 180,E1 16142.037,E2 16142.037} C_VEL
LIN {X 0,Y 377.873,Z 950.759,A -85,B 0,C 180,E1 16141.169,E2 16141.169} C_VEL
LIN {X 0,Y 375.634,Z 968.672,A -85,B 0,C 180,E1 16140.027,E2 16140.027} C_VEL
LIN {X 0,Y 373.231,Z 985.52,A -85,B 0,C 180,E1 16138.654,E2 16138.654} C_VEL
LIN {X 0,Y 370.751,Z 1001.642,A -85,B 0,C 180,E1 16137.02,E2 16137.02} C_VEL
LIN {X 0,Y 368.211,Z 1017.386,A -85,B 0,C 180,E1 16135.062,E2 16135.062} C_VEL
LIN {X 0,Y 365.875,Z 1032.088,A -85,B 0,C 180,E1 16132.833,E2 16132.833} C_VEL
LIN {X 0,Y 363.921,Z 1045.224,A -85,B 0,C 180,E1 16130.421,E2 16130.421} C_VEL
LIN {X 0,Y 362.4,Z 1056.844,A -85,B 0,C 180,E1 16127.833,E2 16127.833} C_VEL
LIN {X 0,Y 361.369,Z 1066.957,A -85,B 0,C 180,E1 16125.075,E2 16125.075} C_VEL
LIN {X 0,Y 360.796,Z 1075.514,A -85,B 0,C 180,E1 16122.158,E2 16122.158} C_VEL
LIN {X 0,Y 360.645,Z 1082.078,A -85,B 0,C 180,E1 16119.253,E2 16119.253} C_VEL
LIN {X 0,Y 360.741,Z 1086.783,A -85,B 0,C 180,E1 16116.365,E2 16116.365} C_VEL
LIN {X 0,Y 360.925,Z 1089.594,A -85,B 0,C 180,E1 16113.653,E2 16113.653} C_VEL
LIN {X 0,Y 361.046,Z 1090.879,A -85,B 0,C 180,E1 16110.952,E2 16110.952} C_VEL
LIN {X 0,Y 361.027,Z 1090.638,A -85,B 0,C 180,E1 16108.254,E2 16108.254} C_VEL
LIN {X 0,Y 360.885,Z 1088.858,A -85,B 0,C 180,E1 16105.55,E2 16105.55} C_VEL
LIN {X 0,Y 360.706,Z 1085.234,A -85,B 0,C 180,E1 16102.674,E2 16102.674} C_VEL
LIN {X 0,Y 360.698,Z 1079.708,A -85,B 0,C 180,E1 16099.757,E2 16099.757} C_VEL
LIN {X 0,Y 360.962,Z 1072.319,A -85,B 0,C 180,E1 16096.871,E2 16096.871} C_VEL
LIN {X 0,Y 361.648,Z 1063.315,A -85,B 0,C 180,E1 16094.114,E2 16094.114} C_VEL
LIN {X 0,Y 362.733,Z 1052.817,A -85,B 0,C 180,E1 16091.518,E2 16091.518} C_VEL
LIN {X 0,Y 364.238,Z 1040.875,A -85,B 0,C 180,E1 16089.092,E2 16089.092} C_VEL
LIN {X 0,Y 366.079,Z 1027.474,A -85,B 0,C 180,E1 16086.839,E2 16086.839} C_VEL
LIN {X 0,Y 368.217,Z 1012.521,A -85,B 0,C 180,E1 16084.765,E2 16084.765} C_VEL
LIN {X 0,Y 370.483,Z 996.54,A -85,B 0,C 180,E1 16082.949,E2 16082.949} C_VEL
LIN {X 0,Y 372.738,Z 979.67,A -85,B 0,C 180,E1 16081.396,E2 16081.396} C_VEL
LIN {X 0,Y 374.903,Z 961.641,A -85,B 0,C 180,E1 16080.084,E2 16080.084} C_VEL
LIN {X 0,Y 376.71,Z 944.082,A -85,B 0,C 180,E1 16079.106,E2 16079.106} C_VEL
LIN {X 0,Y 378.239,Z 925.317,A -85,B 0,C 180,E1 16078.349,E2 16078.349} C_VEL
LIN {X 0,Y 379.15,Z 906.112,A -85,B 0,C 180,E1 16077.843,E2 16077.843} C_VEL
LIN {X 0,Y 382.952,Z 741.978,A -85,B 0,C 180,E1 16074.74,E2 16074.74} C_VEL
LIN {X 0,Y 378.879,Z 706.753,A -85,B 0,C 180,E1 16073.638,E2 16073.638} C_VEL
LIN {X 0,Y 381.635,Z 685.01,A -85,B 0,C 180,E1 16071.232,E2 16071.232} C_VEL
LIN {X 0,Y 374.284,Z 662.966,A -85,B 0,C 180,E1 16067.686,E2 16067.686} C_VEL
LIN {X 0,Y 367.521,Z 644.326,A -85,B 0,C 180,E1 16064.361,E2 16064.361} C_VEL
LIN {X 0,Y 361.83,Z 629.361,A -85,B 0,C 180,E1 16061.37,E2 16061.37} C_VEL
LIN {X 0,Y 361.806,Z 629.169,A -85,B 0,C 180,E1 16057.244,E2 16057.244} C_VEL
LIN {X 0,Y 361.807,Z 629.165,A -85,B 0,C 180,E1 16052.984,E2 16052.984} C_VEL
LIN {X 0,Y 361.813,Z 629.167,A -85,B 0,C 180,E1 16048.74,E2 16048.74} C_VEL
LIN {X 0,Y 361.806,Z 629.166,A -85,B 0,C 180,E1 16044.489,E2 16044.489} C_VEL
LIN {X 0,Y 361.835,Z 629.376,A -85,B 0,C 180,E1 16040.932,E2 16040.932} C_VEL
LIN {X 0,Y 362.521,Z 631.621,A -85,B 0,C 180,E1 16040.322,E2 16040.322} C_VEL
LIN {X 0,Y 364.574,Z 634.963,A -85,B 0,C 180,E1 16039.362,E2 16039.362} C_VEL
LIN {X 0,Y 367.122,Z 640.203,A -85,B 0,C 180,E1 16038.088,E2 16038.088} C_VEL
LIN {X 0,Y 370.297,Z 646.908,A -85,B 0,C 180,E1 16036.552,E2 16036.552} C_VEL
LIN {X 0,Y 374.855,Z 658.531,A -85,B 0,C 180,E1 16034.205,E2 16034.205} C_VEL
LIN {X 0,Y 378.512,Z 670.971,A -85,B 0,C 180,E1 16031.968,E2 16031.968} C_VEL
LIN {X 0,Y 380.141,Z 678.585,A -85,B 0,C 180,E1 16030.763,E2 16030.763} C_VEL
LIN {X 0,Y 378.691,Z 711.407,A -85,B 0,C 180,E1 16026.671,E2 16026.671} C_VEL
LIN {X 0,Y 377.93,Z 727.631,A -85,B 0,C 180,E1 16024.628,E2 16024.628} C_VEL
LIN {X 0,Y 378.225,Z 730.748,A -85,B 0,C 180,E1 16024.491,E2 16024.491} C_VEL
LIN {X 0,Y 373.601,Z 852.777,A -85,B 0,C 180,E1 16021.538,E2 16021.538} C_VEL
LIN {X 0,Y 373.413,Z 871.862,A -85,B 0,C 180,E1 16020.963,E2 16020.963} C_VEL
LIN {X 0,Y 372.899,Z 887.945,A -85,B 0,C 180,E1 16020.196,E2 16020.196} C_VEL
LIN {X 0,Y 371.993,Z 903.565,A -85,B 0,C 180,E1 16019.139,E2 16019.139} C_VEL
LIN {X 0,Y 370.89,Z 917.331,A -85,B 0,C 180,E1 16017.914,E2 16017.914} C_VEL
LIN {X 0,Y 369.53,Z 931.031,A -85,B 0,C 180,E1 16016.354,E2 16016.354} C_VEL
LIN {X 0,Y 368.163,Z 942.53,A -85,B 0,C 180,E1 16014.702,E2 16014.702} C_VEL
LIN {X 0,Y 366.753,Z 953.108,A -85,B 0,C 180,E1 16012.795,E2 16012.795} C_VEL
LIN {X 0,Y 365.428,Z 962.219,A -85,B 0,C 180,E1 16010.71,E2 16010.71} C_VEL
LIN {X 0,Y 364.269,Z 969.862,A -85,B 0,C 180,E1 16008.441,E2 16008.441} C_VEL
LIN {X 0,Y 363.369,Z 975.589,A -85,B 0,C 180,E1 16006.149,E2 16006.149} C_VEL
LIN {X 0,Y 362.65,Z 979.876,A -85,B 0,C 180,E1 16003.633,E2 16003.633} C_VEL
LIN {X 0,Y 362.192,Z 982.239,A -85,B 0,C 180,E1 16001.156,E2 16001.156} C_VEL
LIN {X 0,Y 361.938,Z 982.862,A -85,B 0,C 180,E1 15998.588,E2 15998.588} C_VEL
LIN {X 0,Y 361.868,Z 981.76,A -85,B 0,C 180,E1 15996.146,E2 15996.146} C_VEL
LIN {X 0,Y 361.984,Z 978.676,A -85,B 0,C 180,E1 15993.502,E2 15993.502} C_VEL
LIN {X 0,Y 362.312,Z 973.919,A -85,B 0,C 180,E1 15991.024,E2 15991.024} C_VEL
LIN {X 0,Y 362.864,Z 967.385,A -85,B 0,C 180,E1 15988.615,E2 15988.615} C_VEL
LIN {X 0,Y 363.575,Z 959.593,A -85,B 0,C 180,E1 15986.437,E2 15986.437} C_VEL
LIN {X 0,Y 364.543,Z 949.634,A -85,B 0,C 180,E1 15984.252,E2 15984.252} C_VEL
LIN {X 0,Y 365.599,Z 938.589,A -85,B 0,C 180,E1 15982.333,E2 15982.333} C_VEL
LIN {X 0,Y 366.755,Z 925.925,A -85,B 0,C 180,E1 15980.564,E2 15980.564} C_VEL
LIN {X 0,Y 367.863,Z 911.804,A -85,B 0,C 180,E1 15979.007,E2 15979.007} C_VEL
LIN {X 0,Y 368.848,Z 897.124,A -85,B 0,C 180,E1 15977.735,E2 15977.735} C_VEL
LIN {X 0,Y 369.661,Z 880.978,A -85,B 0,C 180,E1 15976.686,E2 15976.686} C_VEL
LIN {X 0,Y 370.166,Z 864.916,A -85,B 0,C 180,E1 15975.943,E2 15975.943} C_VEL
LIN {X 0,Y 370.387,Z 846.365,A -85,B 0,C 180,E1 15975.413,E2 15975.413} C_VEL
LIN {X 0,Y 373.366,Z 724.073,A -85,B 0,C 180,E1 15972.703,E2 15972.703} C_VEL
LIN {X 0,Y 371.964,Z 715.671,A -85,B 0,C 180,E1 15972.374,E2 15972.374} C_VEL
LIN {X 0,Y 373.2,Z 684.888,A -85,B 0,C 180,E1 15968.431,E2 15968.431} C_VEL
LIN {X 0,Y 373.604,Z 669.557,A -85,B 0,C 180,E1 15966.451,E2 15966.451} C_VEL
LIN {X 0,Y 368.988,Z 652.135,A -85,B 0,C 180,E1 15963.745,E2 15963.745} C_VEL
LIN {X 0,Y 363.423,Z 634.383,A -85,B 0,C 180,E1 15960.864,E2 15960.864} C_VEL
LIN {X 0,Y 361.798,Z 629.362,A -85,B 0,C 180,E1 15959.969,E2 15959.969} C_VEL
LIN {X 0,Y 361.763,Z 629.135,A -85,B 0,C 180,E1 15955.893,E2 15955.893} C_VEL
LIN {X 0,Y 361.771,Z 629.26,A -85,B 0,C 180,E1 15954.406,E2 15954.406} C_VEL
LIN {X 0,Y 362.944,Z 632.866,A -85,B 0,C 180,E1 15953.455,E2 15953.455} C_VEL
LIN {X 0,Y 367.67,Z 647.611,A -85,B 0,C 180,E1 15950.039,E2 15950.039} C_VEL
LIN {X 0,Y 372.295,Z 664.196,A -85,B 0,C 180,E1 15946.506,E2 15946.506} C_VEL
LIN {X 0,Y 374.807,Z 675.106,A -85,B 0,C 180,E1 15944.286,E2 15944.286} C_VEL
LIN {X 0,Y 372.504,Z 694.839,A -85,B 0,C 180,E1 15941.058,E2 15941.058} C_VEL
LIN {X 0,Y 373.17,Z 697.08,A -85,B 0,C 180,E1 15940.83,E2 15940.83} C_VEL
LIN {X 0,Y 376.992,Z 704.464,A -85,B 0,C 180,E1 15940.365,E2 15940.365} C_VEL
LIN {X 0,Y 378.035,Z 708.894,A -85,B 0,C 180,E1 15940.178,E2 15940.178} C_VEL
LIN {X 0,Y 377.999,Z 712.471,A -85,B 0,C 180,E1 15940.125,E2 15940.125} C_VEL
LIN {X 0,Y 376.566,Z 717.244,A -85,B 0,C 180,E1 15940.172,E2 15940.172} C_VEL
LIN {X 0,Y 372.331,Z 726.366,A -85,B 0,C 180,E1 15940.282,E2 15940.282} C_VEL
LIN {X 0,Y 371.664,Z 730.011,A -85,B 0,C 180,E1 15940.249,E2 15940.249} C_VEL
LIN {X 0,Y 368.605,Z 849.946,A -85,B 0,C 180,E1 15937.849,E2 15937.849} C_VEL
LIN {X 0,Y 367.883,Z 867.234,A -85,B 0,C 180,E1 15937.207,E2 15937.207} C_VEL
LIN {X 0,Y 366.829,Z 883.178,A -85,B 0,C 180,E1 15936.338,E2 15936.338} C_VEL
LIN {X 0,Y 365.477,Z 898.229,A -85,B 0,C 180,E1 15935.237,E2 15935.237} C_VEL
LIN {X 0,Y 363.758,Z 913.455,A -85,B 0,C 180,E1 15933.783,E2 15933.783} C_VEL
LIN {X 0,Y 362.002,Z 927.088,A -85,B 0,C 180,E1 15932.137,E2 15932.137} C_VEL
LIN {X 0,Y 360.272,Z 939.15,A -85,B 0,C 180,E1 15930.318,E2 15930.318} C_VEL
LIN {X 0,Y 358.564,Z 950.204,A -85,B 0,C 180,E1 15928.243,E2 15928.243} C_VEL
LIN {X 0,Y 357.055,Z 959.831,A -85,B 0,C 180,E1 15925.986,E2 15925.986} C_VEL
LIN {X 0,Y 355.802,Z 967.947,A -85,B 0,C 180,E1 15923.546,E2 15923.546} C_VEL
LIN {X 0,Y 354.865,Z 974.528,A -85,B 0,C 180,E1 15920.922,E2 15920.922} C_VEL
LIN {X 0,Y 354.276,Z 979.277,A -85,B 0,C 180,E1 15918.276,E2 15918.276} C_VEL
LIN {X 0,Y 353.971,Z 982.246,A -85,B 0,C 180,E1 15915.607,E2 15915.607} C_VEL
LIN {X 0,Y 353.939,Z 983.629,A -85,B 0,C 180,E1 15912.715,E2 15912.715} C_VEL
LIN {X 0,Y 354.178,Z 983.262,A -85,B 0,C 180,E1 15910.027,E2 15910.027} C_VEL
LIN {X 0,Y 354.746,Z 981.013,A -85,B 0,C 180,E1 15907.17,E2 15907.17} C_VEL
LIN {X 0,Y 355.7,Z 976.919,A -85,B 0,C 180,E1 15904.349,E2 15904.349} C_VEL
LIN {X 0,Y 356.996,Z 971.27,A -85,B 0,C 180,E1 15901.75,E2 15901.75} C_VEL
LIN {X 0,Y 358.762,Z 963.534,A -85,B 0,C 180,E1 15899.15,E2 15899.15} C_VEL
LIN {X 0,Y 360.8,Z 954.522,A -85,B 0,C 180,E1 15896.816,E2 15896.816} C_VEL
LIN {X 0,Y 363.04,Z 943.909,A -85,B 0,C 180,E1 15894.665,E2 15894.665} C_VEL
LIN {X 0,Y 365.448,Z 931.582,A -85,B 0,C 180,E1 15892.673,E2 15892.673} C_VEL
LIN {X 0,Y 367.726,Z 918.64,A -85,B 0,C 180,E1 15891,E2 15891} C_VEL
LIN {X 0,Y 369.843,Z 904.394,A -85,B 0,C 180,E1 15889.547,E2 15889.547} C_VEL
LIN {X 0,Y 371.682,Z 889.53,A -85,B 0,C 180,E1 15888.36,E2 15888.36} C_VEL
LIN {X 0,Y 373.204,Z 873.363,A -85,B 0,C 180,E1 15887.385,E2 15887.385} C_VEL
LIN {X 0,Y 374.194,Z 856.552,A -85,B 0,C 180,E1 15886.683,E2 15886.683} C_VEL
LIN {X 0,Y 374.86,Z 834.787,A -85,B 0,C 180,E1 15886.14,E2 15886.14} C_VEL
LIN {X 0,Y 378.191,Z 731.322,A -85,B 0,C 180,E1 15884.039,E2 15884.039} C_VEL
LIN {X 0,Y 371.654,Z 701.892,A -85,B 0,C 180,E1 15882.54,E2 15882.54} C_VEL
LIN {X 0,Y 370.438,Z 696.289,A -85,B 0,C 180,E1 15882.185,E2 15882.185} C_VEL
LIN {X 0,Y 372.003,Z 685.085,A -85,B 0,C 180,E1 15880.242,E2 15880.242} C_VEL
LIN {X 0,Y 368.827,Z 672.18,A -85,B 0,C 180,E1 15877.155,E2 15877.155} C_VEL
LIN {X 0,Y 365.021,Z 659.521,A -85,B 0,C 180,E1 15873.784,E2 15873.784} C_VEL
LIN {X 0,Y 361.051,Z 648.159,A -85,B 0,C 180,E1 15870.45,E2 15870.45} C_VEL
LIN {X 0,Y 356.929,Z 637.695,A -85,B 0,C 180,E1 15866.989,E2 15866.989} C_VEL
LIN {X 0,Y 353.879,Z 630.251,A -85,B 0,C 180,E1 15864.132,E2 15864.132} C_VEL
LIN {X 0,Y 353.866,Z 630.153,A -85,B 0,C 180,E1 15859.992,E2 15859.992} C_VEL
LIN {X 0,Y 353.866,Z 630.147,A -85,B 0,C 180,E1 15855.739,E2 15855.739} C_VEL
LIN {X 0,Y 353.862,Z 630.149,A -85,B 0,C 180,E1 15851.573,E2 15851.573} C_VEL
LIN {X 0,Y 353.867,Z 630.153,A -85,B 0,C 180,E1 15847.305,E2 15847.305} C_VEL
LIN {X 0,Y 353.86,Z 630.159,A -85,B 0,C 180,E1 15843.078,E2 15843.078} C_VEL
LIN {X 0,Y 353.862,Z 630.15,A -85,B 0,C 180,E1 15838.867,E2 15838.867} C_VEL
LIN {X 0,Y 353.855,Z 630.136,A -85,B 0,C 180,E1 15834.65,E2 15834.65} C_VEL
LIN {X 0,Y 353.857,Z 630.13,A -85,B 0,C 180,E1 15830.568,E2 15830.568} C_VEL
LIN {X 0,Y 353.86,Z 630.132,A -85,B 0,C 180,E1 15826.408,E2 15826.408} C_VEL
LIN {X 0,Y 353.858,Z 630.138,A -85,B 0,C 180,E1 15822.217,E2 15822.217} C_VEL
LIN {X 0,Y 353.863,Z 630.145,A -85,B 0,C 180,E1 15818.101,E2 15818.101} C_VEL
LIN {X 0,Y 353.856,Z 630.147,A -85,B 0,C 180,E1 15813.846,E2 15813.846} C_VEL
LIN {X 0,Y 353.856,Z 630.144,A -85,B 0,C 180,E1 15809.617,E2 15809.617} C_VEL
LIN {X 0,Y 353.852,Z 630.142,A -85,B 0,C 180,E1 15805.393,E2 15805.393} C_VEL
LIN {X 0,Y 353.911,Z 630.531,A -85,B 0,C 180,E1 15804.733,E2 15804.733} C_VEL
LIN {X 0,Y 355.664,Z 634.334,A -85,B 0,C 180,E1 15803.417,E2 15803.417} C_VEL
LIN {X 0,Y 358.386,Z 640.448,A -85,B 0,C 180,E1 15801.527,E2 15801.527} C_VEL
LIN {X 0,Y 361.663,Z 647.444,A -85,B 0,C 180,E1 15799.482,E2 15799.482} C_VEL
LIN {X 0,Y 366.75,Z 659.579,A -85,B 0,C 180,E1 15796.39,E2 15796.39} C_VEL
LIN {X 0,Y 371.776,Z 672.808,A -85,B 0,C 180,E1 15793.436,E2 15793.436} C_VEL
LIN {X 0,Y 376.378,Z 686.979,A -85,B 0,C 180,E1 15790.673,E2 15790.673} C_VEL
LIN {X 0,Y 377.657,Z 691.956,A -85,B 0,C 180,E1 15789.794,E2 15789.794} C_VEL
LIN {X 0,Y 375.235,Z 706.883,A -85,B 0,C 180,E1 15788.067,E2 15788.067} C_VEL
LIN {X 0,Y 379.141,Z 740.181,A -85,B 0,C 180,E1 15786.814,E2 15786.814} C_VEL
LIN {X 0,Y 379.573,Z 747.326,A -85,B 0,C 180,E1 15786.597,E2 15786.597} C_VEL
LIN {X 0,Y 374.42,Z 912.529,A -85,B 0,C 180,E1 15783.315,E2 15783.315} C_VEL
LIN {X 0,Y 372.961,Z 931.644,A -85,B 0,C 180,E1 15782.684,E2 15782.684} C_VEL
LIN {X 0,Y 371.109,Z 948.747,A -85,B 0,C 180,E1 15781.875,E2 15781.875} C_VEL
LIN {X 0,Y 368.77,Z 966.584,A -85,B 0,C 180,E1 15780.741,E2 15780.741} C_VEL
LIN {X 0,Y 366.221,Z 983.644,A -85,B 0,C 180,E1 15779.345,E2 15779.345} C_VEL
LIN {X 0,Y 363.567,Z 999.931,A -85,B 0,C 180,E1 15777.682,E2 15777.682} C_VEL
LIN {X 0,Y 360.973,Z 1015.165,A -85,B 0,C 180,E1 15775.777,E2 15775.777} C_VEL
LIN {X 0,Y 358.62,Z 1029.076,A -85,B 0,C 180,E1 15773.671,E2 15773.671} C_VEL
LIN {X 0,Y 356.46,Z 1042.488,A -85,B 0,C 180,E1 15771.213,E2 15771.213} C_VEL
LIN {X 0,Y 354.751,Z 1054.356,A -85,B 0,C 180,E1 15768.571,E2 15768.571} C_VEL
LIN {X 0,Y 353.567,Z 1064.715,A -85,B 0,C 180,E1 15765.752,E2 15765.752} C_VEL
LIN {X 0,Y 352.906,Z 1073.049,A -85,B 0,C 180,E1 15762.933,E2 15762.933} C_VEL
LIN {X 0,Y 352.688,Z 1079.921,A -85,B 0,C 180,E1 15759.958,E2 15759.958} C_VEL
LIN {X 0,Y 352.758,Z 1084.925,A -85,B 0,C 180,E1 15757,E2 15757} C_VEL
LIN {X 0,Y 352.974,Z 1088.161,A -85,B 0,C 180,E1 15754.06,E2 15754.06} C_VEL
LIN {X 0,Y 353.129,Z 1089.661,A -85,B 0,C 180,E1 15751.135,E2 15751.135} C_VEL
LIN {X 0,Y 353.118,Z 1089.495,A -85,B 0,C 180,E1 15748.377,E2 15748.377} C_VEL
LIN {X 0,Y 352.966,Z 1087.78,A -85,B 0,C 180,E1 15745.613,E2 15745.613} C_VEL
LIN {X 0,Y 352.766,Z 1084.207,A -85,B 0,C 180,E1 15742.672,E2 15742.672} C_VEL
LIN {X 0,Y 352.739,Z 1078.79,A -85,B 0,C 180,E1 15739.713,E2 15739.713} C_VEL
LIN {X 0,Y 353.002,Z 1071.393,A -85,B 0,C 180,E1 15736.736,E2 15736.736} C_VEL
LIN {X 0,Y 353.712,Z 1062.42,A -85,B 0,C 180,E1 15733.917,E2 15733.917} C_VEL
LIN {X 0,Y 354.867,Z 1051.711,A -85,B 0,C 180,E1 15731.208,E2 15731.208} C_VEL
LIN {X 0,Y 356.407,Z 1040.056,A -85,B 0,C 180,E1 15728.783,E2 15728.783} C_VEL
LIN {X 0,Y 358.33,Z 1026.703,A -85,B 0,C 180,E1 15726.483,E2 15726.483} C_VEL
LIN {X 0,Y 360.453,Z 1012.491,A -85,B 0,C 180,E1 15724.457,E2 15724.457} C_VEL
LIN {X 0,Y 362.801,Z 996.604,A -85,B 0,C 180,E1 15722.597,E2 15722.597} C_VEL
LIN {X 0,Y 365.139,Z 979.853,A -85,B 0,C 180,E1 15721.008,E2 15721.008} C_VEL
LIN {X 0,Y 367.365,Z 962.157,A -85,B 0,C 180,E1 15719.676,E2 15719.676} C_VEL
LIN {X 0,Y 369.332,Z 943.955,A -85,B 0,C 180,E1 15718.628,E2 15718.628} C_VEL
LIN {X 0,Y 370.953,Z 924.93,A -85,B 0,C 180,E1 15717.839,E2 15717.839} C_VEL
LIN {X 0,Y 371.903,Z 905.788,A -85,B 0,C 180,E1 15717.321,E2 15717.321} C_VEL
LIN {X 0,Y 375.874,Z 743.08,A -85,B 0,C 180,E1 15714.196,E2 15714.196} C_VEL
LIN {X 0,Y 371.757,Z 706.441,A -85,B 0,C 180,E1 15713.015,E2 15713.015} C_VEL
LIN {X 0,Y 374.31,Z 687.785,A -85,B 0,C 180,E1 15710.919,E2 15710.919} C_VEL
LIN {X 0,Y 367.157,Z 666.022,A -85,B 0,C 180,E1 15707.33,E2 15707.33} C_VEL
LIN {X 0,Y 360.2,Z 646.673,A -85,B 0,C 180,E1 15703.803,E2 15703.803} C_VEL
LIN {X 0,Y 353.889,Z 630.338,A -85,B 0,C 180,E1 15700.41,E2 15700.41} C_VEL
LIN {X 0,Y 353.859,Z 630.155,A -85,B 0,C 180,E1 15696.361,E2 15696.361} C_VEL
LIN {X 0,Y 353.856,Z 630.159,A -85,B 0,C 180,E1 15692.087,E2 15692.087} C_VEL
LIN {X 0,Y 353.853,Z 630.156,A -85,B 0,C 180,E1 15687.79,E2 15687.79} C_VEL
LIN {X 0,Y 353.846,Z 630.161,A -85,B 0,C 180,E1 15683.656,E2 15683.656} C_VEL
LIN {X 0,Y 353.925,Z 630.499,A -85,B 0,C 180,E1 15682.77,E2 15682.77} C_VEL
LIN {X 0,Y 355.571,Z 634.211,A -85,B 0,C 180,E1 15681.615,E2 15681.615} C_VEL
LIN {X 0,Y 356.9,Z 635.955,A -85,B 0,C 180,E1 15681.014,E2 15681.014} C_VEL
LIN {X 0,Y 358.666,Z 639.479,A -85,B 0,C 180,E1 15680.037,E2 15680.037} C_VEL
LIN {X 0,Y 361.811,Z 645.94,A -85,B 0,C 180,E1 15678.363,E2 15678.363} C_VEL
LIN {X 0,Y 365.981,Z 655.323,A -85,B 0,C 180,E1 15676.18,E2 15676.18} C_VEL
LIN {X 0,Y 370.137,Z 667.508,A -85,B 0,C 180,E1 15673.752,E2 15673.752} C_VEL
LIN {X 0,Y 373.309,Z 679.86,A -85,B 0,C 180,E1 15671.588,E2 15671.588} C_VEL
LIN {X 0,Y 373.54,Z 683.122,A -85,B 0,C 180,E1 15671.111,E2 15671.111} C_VEL
LIN {X 0,Y 372.01,Z 714.303,A -85,B 0,C 180,E1 15667.179,E2 15667.179} C_VEL
LIN {X 0,Y 371.263,Z 729.197,A -85,B 0,C 180,E1 15665.292,E2 15665.292} C_VEL
LIN {X 0,Y 371.572,Z 732.239,A -85,B 0,C 180,E1 15665.152,E2 15665.152} C_VEL
LIN {X 0,Y 366.609,Z 853.083,A -85,B 0,C 180,E1 15662.139,E2 15662.139} C_VEL
LIN {X 0,Y 366.362,Z 872.998,A -85,B 0,C 180,E1 15661.524,E2 15661.524} C_VEL
LIN {X 0,Y 365.836,Z 888.356,A -85,B 0,C 180,E1 15660.783,E2 15660.783} C_VEL
LIN {X 0,Y 364.908,Z 903.846,A -85,B 0,C 180,E1 15659.737,E2 15659.737} C_VEL
LIN {X 0,Y 363.755,Z 917.851,A -85,B 0,C 180,E1 15658.495,E2 15658.495} C_VEL
LIN {X 0,Y 362.299,Z 931.601,A -85,B 0,C 180,E1 15656.915,E2 15656.915} C_VEL
LIN {X 0,Y 360.839,Z 943.252,A -85,B 0,C 180,E1 15655.231,E2 15655.231} C_VEL
LIN {X 0,Y 359.205,Z 954.735,A -85,B 0,C 180,E1 15653.125,E2 15653.125} C_VEL
LIN {X 0,Y 357.794,Z 963.788,A -85,B 0,C 180,E1 15650.996,E2 15650.996} C_VEL
LIN {X 0,Y 356.555,Z 971.375,A -85,B 0,C 180,E1 15648.679,E2 15648.679} C_VEL
LIN {X 0,Y 355.583,Z 977.018,A -85,B 0,C 180,E1 15646.337,E2 15646.337} C_VEL
LIN {X 0,Y 354.816,Z 981.206,A -85,B 0,C 180,E1 15643.8,E2 15643.8} C_VEL
LIN {X 0,Y 354.313,Z 983.551,A -85,B 0,C 180,E1 15641.234,E2 15641.234} C_VEL
LIN {X 0,Y 354.038,Z 984.113,A -85,B 0,C 180,E1 15638.634,E2 15638.634} C_VEL
LIN {X 0,Y 353.956,Z 982.982,A -85,B 0,C 180,E1 15636.174,E2 15636.174} C_VEL
LIN {X 0,Y 354.07,Z 979.906,A -85,B 0,C 180,E1 15633.501,E2 15633.501} C_VEL
LIN {X 0,Y 354.401,Z 975.199,A -85,B 0,C 180,E1 15630.998,E2 15630.998} C_VEL
LIN {X 0,Y 354.953,Z 968.837,A -85,B 0,C 180,E1 15628.592,E2 15628.592} C_VEL
LIN {X 0,Y 355.71,Z 960.874,A -85,B 0,C 180,E1 15626.308,E2 15626.308} C_VEL
LIN {X 0,Y 356.697,Z 951.07,A -85,B 0,C 180,E1 15624.106,E2 15624.106} C_VEL
LIN {X 0,Y 357.782,Z 940.186,A -85,B 0,C 180,E1 15622.163,E2 15622.163} C_VEL
LIN {X 0,Y 359.02,Z 927.137,A -85,B 0,C 180,E1 15620.296,E2 15620.296} C_VEL
LIN {X 0,Y 360.135,Z 913.52,A -85,B 0,C 180,E1 15618.757,E2 15618.757} C_VEL
LIN {X 0,Y 361.191,Z 898.541,A -85,B 0,C 180,E1 15617.422,E2 15617.422} C_VEL
LIN {X 0,Y 362.047,Z 882.235,A -85,B 0,C 180,E1 15616.336,E2 15616.336} C_VEL
LIN {X 0,Y 362.587,Z 865.903,A -85,B 0,C 180,E1 15615.563,E2 15615.563} C_VEL
LIN {X 0,Y 362.826,Z 847.155,A -85,B 0,C 180,E1 15615.015,E2 15615.015} C_VEL
LIN {X 0,Y 365.97,Z 725.185,A -85,B 0,C 180,E1 15612.243,E2 15612.243} C_VEL
LIN {X 0,Y 364.566,Z 716.614,A -85,B 0,C 180,E1 15611.9,E2 15611.9} C_VEL
LIN {X 0,Y 365.933,Z 684.381,A -85,B 0,C 180,E1 15607.738,E2 15607.738} C_VEL
LIN {X 0,Y 366.229,Z 672.074,A -85,B 0,C 180,E1 15606.137,E2 15606.137} C_VEL
LIN {X 0,Y 361.51,Z 654.372,A -85,B 0,C 180,E1 15603.356,E2 15603.356} C_VEL
LIN {X 0,Y 356.132,Z 637.296,A -85,B 0,C 180,E1 15600.542,E2 15600.542} C_VEL
LIN {X 0,Y 353.884,Z 630.341,A -85,B 0,C 180,E1 15599.308,E2 15599.308} C_VEL
LIN {X 0,Y 353.872,Z 630.259,A -85,B 0,C 180,E1 15595.289,E2 15595.289} C_VEL
LIN {X 0,Y 355.281,Z 634.825,A -85,B 0,C 180,E1 15594.084,E2 15594.084} C_VEL
LIN {X 0,Y 359.937,Z 649.17,A -85,B 0,C 180,E1 15590.659,E2 15590.659} C_VEL
LIN {X 0,Y 364.334,Z 664.713,A -85,B 0,C 180,E1 15587.241,E2 15587.241} C_VEL
LIN {X 0,Y 367.383,Z 677.567,A -85,B 0,C 180,E1 15584.581,E2 15584.581} C_VEL
LIN {X 0,Y 365.193,Z 695.444,A -85,B 0,C 180,E1 15581.61,E2 15581.61} C_VEL
LIN {X 0,Y 366.053,Z 700.594,A -85,B 0,C 180,E1 15581.354,E2 15581.354} C_VEL
LIN {X 0,Y 371.664,Z 730.011,A -85,B 0,C 180,E1 15580.249,E2 15580.249} C_VEL
LIN {X 0,Y 370.587,Z 737.686,A -85,B 0,C 180,E1 15580.172,E2 15580.172} C_VEL
LIN {X 0,Y 364.511,Z 758.048,A -85,B 0,C 180,E1 15580.233,E2 15580.233} C_VEL
LIN {X 0,Y 363.675,Z 764.638,A -85,B 0,C 180,E1 15580.158,E2 15580.158} C_VEL
LIN {X 0,Y 361.381,Z 850.996,A -85,B 0,C 180,E1 15578.373,E2 15578.373} C_VEL
LIN {X 0,Y 360.614,Z 868.389,A -85,B 0,C 180,E1 15577.709,E2 15577.709} C_VEL
LIN {X 0,Y 359.475,Z 884.748,A -85,B 0,C 180,E1 15576.792,E2 15576.792} C_VEL
LIN {X 0,Y 357.984,Z 900.271,A -85,B 0,C 180,E1 15575.61,E2 15575.61} C_VEL
LIN {X 0,Y 356.179,Z 915.495,A -85,B 0,C 180,E1 15574.105,E2 15574.105} C_VEL
LIN {X 0,Y 354.361,Z 928.934,A -85,B 0,C 180,E1 15572.426,E2 15572.426} C_VEL
LIN {X 0,Y 352.488,Z 941.273,A -85,B 0,C 180,E1 15570.488,E2 15570.488} C_VEL
LIN {X 0,Y 350.731,Z 952.158,A -85,B 0,C 180,E1 15568.367,E2 15568.367} C_VEL
LIN {X 0,Y 349.185,Z 961.625,A -85,B 0,C 180,E1 15566.06,E2 15566.06} C_VEL
LIN {X 0,Y 347.894,Z 969.575,A -85,B 0,C 180,E1 15563.565,E2 15563.565} C_VEL
LIN {X 0,Y 346.938,Z 976.054,A -85,B 0,C 180,E1 15560.88,E2 15560.88} C_VEL
LIN {X 0,Y 346.338,Z 980.707,A -85,B 0,C 180,E1 15558.148,E2 15558.148} C_VEL
LIN {X 0,Y 346.036,Z 983.675,A -85,B 0,C 180,E1 15555.27,E2 15555.27} C_VEL
LIN {X 0,Y 346.048,Z 984.889,A -85,B 0,C 180,E1 15552.34,E2 15552.34} C_VEL
LIN {X 0,Y 346.345,Z 984.293,A -85,B 0,C 180,E1 15549.555,E2 15549.555} C_VEL
LIN {X 0,Y 347.027,Z 981.801,A -85,B 0,C 180,E1 15546.572,E2 15546.572} C_VEL
LIN {X 0,Y 348.011,Z 977.899,A -85,B 0,C 180,E1 15543.923,E2 15543.923} C_VEL
LIN {X 0,Y 349.42,Z 972.137,A -85,B 0,C 180,E1 15541.267,E2 15541.267} C_VEL
LIN {X 0,Y 351.335,Z 964.327,A -85,B 0,C 180,E1 15538.615,E2 15538.615} C_VEL
LIN {X 0,Y 353.493,Z 955.338,A -85,B 0,C 180,E1 15536.262,E2 15536.262} C_VEL
LIN {X 0,Y 355.908,Z 944.516,A -85,B 0,C 180,E1 15534.046,E2 15534.046} C_VEL
LIN {X 0,Y 358.443,Z 932.248,A -85,B 0,C 180,E1 15532.041,E2 15532.041} C_VEL
LIN {X 0,Y 360.876,Z 919.008,A -85,B 0,C 180,E1 15530.321,E2 15530.321} C_VEL
LIN {X 0,Y 363.113,Z 904.624,A -85,B 0,C 180,E1 15528.845,E2 15528.845} C_VEL
LIN {X 0,Y 365.051,Z 889.583,A -85,B 0,C 180,E1 15527.641,E2 15527.641} C_VEL
LIN {X 0,Y 366.603,Z 873.477,A -85,B 0,C 180,E1 15526.673,E2 15526.673} C_VEL
LIN {X 0,Y 367.64,Z 856.41,A -85,B 0,C 180,E1 15525.963,E2 15525.963} C_VEL
LIN {X 0,Y 368.384,Z 833.262,A -85,B 0,C 180,E1 15525.393,E2 15525.393} C_VEL
LIN {X 0,Y 371.805,Z 732.853,A -85,B 0,C 180,E1 15523.321,E2 15523.321} C_VEL
LIN {X 0,Y 365.474,Z 703.959,A -85,B 0,C 180,E1 15521.799,E2 15521.799} C_VEL
LIN {X 0,Y 363.799,Z 696.484,A -85,B 0,C 180,E1 15521.328,E2 15521.328} C_VEL
LIN {X 0,Y 364.98,Z 688.258,A -85,B 0,C 180,E1 15519.87,E2 15519.87} C_VEL
LIN {X 0,Y 361.873,Z 675.504,A -85,B 0,C 180,E1 15516.749,E2 15516.749} C_VEL
LIN {X 0,Y 358.26,Z 663.388,A -85,B 0,C 180,E1 15513.44,E2 15513.44} C_VEL
LIN {X 0,Y 354.44,Z 652.424,A -85,B 0,C 180,E1 15510.141,E2 15510.141} C_VEL
LIN {X 0,Y 350.643,Z 642.535,A -85,B 0,C 180,E1 15506.779,E2 15506.779} C_VEL
LIN {X 0,Y 347.275,Z 634.699,A -85,B 0,C 180,E1 15503.771,E2 15503.771} C_VEL
LIN {X 0,Y 345.942,Z 631.225,A -85,B 0,C 180,E1 15502.249,E2 15502.249} C_VEL
LIN {X 0,Y 345.925,Z 631.127,A -85,B 0,C 180,E1 15498.016,E2 15498.016} C_VEL
LIN {X 0,Y 345.928,Z 631.126,A -85,B 0,C 180,E1 15493.71,E2 15493.71} C_VEL
LIN {X 0,Y 345.923,Z 631.124,A -85,B 0,C 180,E1 15489.483,E2 15489.483} C_VEL
LIN {X 0,Y 345.921,Z 631.121,A -85,B 0,C 180,E1 15485.307,E2 15485.307} C_VEL
LIN {X 0,Y 345.921,Z 631.12,A -85,B 0,C 180,E1 15480.994,E2 15480.994} C_VEL
LIN {X 0,Y 345.917,Z 631.125,A -85,B 0,C 180,E1 15476.852,E2 15476.852} C_VEL
LIN {X 0,Y 345.919,Z 631.135,A -85,B 0,C 180,E1 15472.527,E2 15472.527} C_VEL
LIN {X 0,Y 345.916,Z 631.144,A -85,B 0,C 180,E1 15468.158,E2 15468.158} C_VEL
LIN {X 0,Y 345.915,Z 631.147,A -85,B 0,C 180,E1 15463.89,E2 15463.89} C_VEL
LIN {X 0,Y 345.916,Z 631.141,A -85,B 0,C 180,E1 15459.528,E2 15459.528} C_VEL
LIN {X 0,Y 345.916,Z 631.14,A -85,B 0,C 180,E1 15455.221,E2 15455.221} C_VEL
LIN {X 0,Y 345.921,Z 631.143,A -85,B 0,C 180,E1 15450.949,E2 15450.949} C_VEL
LIN {X 0,Y 345.939,Z 631.293,A -85,B 0,C 180,E1 15446.746,E2 15446.746} C_VEL
LIN {X 0,Y 347.567,Z 635.105,A -85,B 0,C 180,E1 15445.278,E2 15445.278} C_VEL
LIN {X 0,Y 350.419,Z 641.142,A -85,B 0,C 180,E1 15443.188,E2 15443.188} C_VEL
LIN {X 0,Y 354.154,Z 649.197,A -85,B 0,C 180,E1 15440.675,E2 15440.675} C_VEL
LIN {X 0,Y 358.685,Z 659.684,A -85,B 0,C 180,E1 15437.794,E2 15437.794} C_VEL
LIN {X 0,Y 363.821,Z 673.018,A -85,B 0,C 180,E1 15434.62,E2 15434.62} C_VEL
LIN {X 0,Y 368.491,Z 686.901,A -85,B 0,C 180,E1 15431.74,E2 15431.74} C_VEL
LIN {X 0,Y 370.683,Z 695.073,A -85,B 0,C 180,E1 15430.24,E2 15430.24} C_VEL
LIN {X 0,Y 368.701,Z 706.329,A -85,B 0,C 180,E1 15428.895,E2 15428.895} C_VEL
LIN {X 0,Y 372.541,Z 739.611,A -85,B 0,C 180,E1 15427.578,E2 15427.578} C_VEL
LIN {X 0,Y 373.097,Z 748.216,A -85,B 0,C 180,E1 15427.303,E2 15427.303} C_VEL
LIN {X 0,Y 367.71,Z 911.703,A -85,B 0,C 180,E1 15424.001,E2 15424.001} C_VEL
LIN {X 0,Y 366.187,Z 930.768,A -85,B 0,C 180,E1 15423.362,E2 15423.362} C_VEL
LIN {X 0,Y 364.09,Z 949.091,A -85,B 0,C 180,E1 15422.471,E2 15422.471} C_VEL
LIN {X 0,Y 361.645,Z 966.703,A -85,B 0,C 180,E1 15421.317,E2 15421.317} C_VEL
LIN {X 0,Y 358.991,Z 983.506,A -85,B 0,C 180,E1 15419.904,E2 15419.904} C_VEL
LIN {X 0,Y 356.147,Z 999.972,A -85,B 0,C 180,E1 15418.172,E2 15418.172} C_VEL
LIN {X 0,Y 353.25,Z 1015.987,A -85,B 0,C 180,E1 15416.09,E2 15416.09} C_VEL
LIN {X 0,Y 350.748,Z 1029.927,A -85,B 0,C 180,E1 15413.878,E2 15413.878} C_VEL
LIN {X 0,Y 348.525,Z 1043.018,A -85,B 0,C 180,E1 15411.367,E2 15411.367} C_VEL
LIN {X 0,Y 346.772,Z 1054.6,A -85,B 0,C 180,E1 15408.666,E2 15408.666} C_VEL
LIN {X 0,Y 345.566,Z 1064.682,A -85,B 0,C 180,E1 15405.782,E2 15405.782} C_VEL
LIN {X 0,Y 344.888,Z 1073.219,A -85,B 0,C 180,E1 15402.728,E2 15402.728} C_VEL
LIN {X 0,Y 344.71,Z 1079.768,A -85,B 0,C 180,E1 15399.685,E2 15399.685} C_VEL
LIN {X 0,Y 344.831,Z 1084.458,A -85,B 0,C 180,E1 15396.66,E2 15396.66} C_VEL
LIN {X 0,Y 345.062,Z 1087.251,A -85,B 0,C 180,E1 15393.821,E2 15393.821} C_VEL
LIN {X 0,Y 345.22,Z 1088.505,A -85,B 0,C 180,E1 15390.995,E2 15390.995} C_VEL
LIN {X 0,Y 345.203,Z 1088.212,A -85,B 0,C 180,E1 15388.174,E2 15388.174} C_VEL
LIN {X 0,Y 345.023,Z 1086.358,A -85,B 0,C 180,E1 15385.345,E2 15385.345} C_VEL
LIN {X 0,Y 344.822,Z 1082.911,A -85,B 0,C 180,E1 15382.502,E2 15382.502} C_VEL
LIN {X 0,Y 344.788,Z 1077.359,A -85,B 0,C 180,E1 15379.442,E2 15379.442} C_VEL
LIN {X 0,Y 345.078,Z 1069.952,A -85,B 0,C 180,E1 15376.426,E2 15376.426} C_VEL
LIN {X 0,Y 345.836,Z 1060.9,A -85,B 0,C 180,E1 15373.54,E2 15373.54} C_VEL
LIN {X 0,Y 347.042,Z 1050.342,A -85,B 0,C 180,E1 15370.825,E2 15370.825} C_VEL
LIN {X 0,Y 348.726,Z 1038.221,A -85,B 0,C 180,E1 15368.274,E2 15368.274} C_VEL
LIN {X 0,Y 350.801,Z 1024.506,A -85,B 0,C 180,E1 15365.897,E2 15365.897} C_VEL
LIN {X 0,Y 353.218,Z 1009.062,A -85,B 0,C 180,E1 15363.704,E2 15363.704} C_VEL
LIN {X 0,Y 355.597,Z 993.536,A -85,B 0,C 180,E1 15361.902,E2 15361.902} C_VEL
LIN {X 0,Y 357.933,Z 977.258,A -85,B 0,C 180,E1 15360.367,E2 15360.367} C_VEL
LIN {X 0,Y 360.183,Z 959.927,A -85,B 0,C 180,E1 15359.067,E2 15359.067} C_VEL
LIN {X 0,Y 362.155,Z 942.01,A -85,B 0,C 180,E1 15358.04,E2 15358.04} C_VEL
LIN {X 0,Y 363.793,Z 923.204,A -85,B 0,C 180,E1 15357.265,E2 15357.265} C_VEL
LIN {X 0,Y 364.725,Z 904.029,A -85,B 0,C 180,E1 15356.75,E2 15356.75} C_VEL
LIN {X 0,Y 368.805,Z 744.008,A -85,B 0,C 180,E1 15353.628,E2 15353.628} C_VEL
LIN {X 0,Y 364.638,Z 706.46,A -85,B 0,C 180,E1 15352.402,E2 15352.402} C_VEL
LIN {X 0,Y 366.795,Z 689.855,A -85,B 0,C 180,E1 15350.483,E2 15350.483} C_VEL
LIN {X 0,Y 359.845,Z 668.606,A -85,B 0,C 180,E1 15346.879,E2 15346.879} C_VEL
LIN {X 0,Y 353.262,Z 650.227,A -85,B 0,C 180,E1 15343.454,E2 15343.454} C_VEL
LIN {X 0,Y 347.156,Z 634.548,A -85,B 0,C 180,E1 15340.177,E2 15340.177} C_VEL
LIN {X 0,Y 345.949,Z 631.313,A -85,B 0,C 180,E1 15339.381,E2 15339.381} C_VEL
LIN {X 0,Y 345.927,Z 631.144,A -85,B 0,C 180,E1 15335.112,E2 15335.112} C_VEL
LIN {X 0,Y 345.934,Z 631.143,A -85,B 0,C 180,E1 15330.769,E2 15330.769} C_VEL
LIN {X 0,Y 345.929,Z 631.145,A -85,B 0,C 180,E1 15326.615,E2 15326.615} C_VEL
LIN {X 0,Y 345.958,Z 631.395,A -85,B 0,C 180,E1 15325.228,E2 15325.228} C_VEL
LIN {X 0,Y 347.003,Z 634.287,A -85,B 0,C 180,E1 15324.152,E2 15324.152} C_VEL
LIN {X 0,Y 349.23,Z 637.115,A -85,B 0,C 180,E1 15322.915,E2 15322.915} C_VEL
LIN {X 0,Y 351.105,Z 640.827,A -85,B 0,C 180,E1 15321.728,E2 15321.728} C_VEL
LIN {X 0,Y 351.95,Z 642.153,A -85,B 0,C 180,E1 15321.278,E2 15321.278} C_VEL
LIN {X 0,Y 355.947,Z 650.144,A -85,B 0,C 180,E1 15319.017,E2 15319.017} C_VEL
LIN {X 0,Y 360.594,Z 661.262,A -85,B 0,C 180,E1 15316.382,E2 15316.382} C_VEL
LIN {X 0,Y 364.448,Z 673.093,A -85,B 0,C 180,E1 15313.97,E2 15313.97} C_VEL
LIN {X 0,Y 367.248,Z 685.033,A -85,B 0,C 180,E1 15311.842,E2 15311.842} C_VEL
LIN {X 0,Y 365.493,Z 716.165,A -85,B 0,C 180,E1 15307.861,E2 15307.861} C_VEL
LIN {X 0,Y 364.689,Z 730.873,A -85,B 0,C 180,E1 15305.98,E2 15305.98} C_VEL
LIN {X 0,Y 364.988,Z 734.018,A -85,B 0,C 180,E1 15305.837,E2 15305.837} C_VEL
LIN {X 0,Y 359.647,Z 855.015,A -85,B 0,C 180,E1 15302.724,E2 15302.724} C_VEL
LIN {X 0,Y 359.383,Z 874.573,A -85,B 0,C 180,E1 15302.102,E2 15302.102} C_VEL
LIN {X 0,Y 358.793,Z 890.381,A -85,B 0,C 180,E1 15301.317,E2 15301.317} C_VEL
LIN {X 0,Y 357.777,Z 905.766,A -85,B 0,C 180,E1 15300.24,E2 15300.24} C_VEL
LIN {X 0,Y 356.518,Z 919.768,A -85,B 0,C 180,E1 15298.955,E2 15298.955} C_VEL
LIN {X 0,Y 354.895,Z 934.098,A -85,B 0,C 180,E1 15297.254,E2 15297.254} C_VEL
LIN {X 0,Y 353.273,Z 945.989,A -85,B 0,C 180,E1 15295.454,E2 15295.454} C_VEL
LIN {X 0,Y 351.682,Z 956.424,A -85,B 0,C 180,E1 15293.47,E2 15293.47} C_VEL
LIN {X 0,Y 350.171,Z 965.366,A -85,B 0,C 180,E1 15291.295,E2 15291.295} C_VEL
LIN {X 0,Y 348.85,Z 972.904,A -85,B 0,C 180,E1 15288.928,E2 15288.928} C_VEL
LIN {X 0,Y 347.808,Z 978.483,A -85,B 0,C 180,E1 15286.534,E2 15286.534} C_VEL
LIN {X 0,Y 346.983,Z 982.607,A -85,B 0,C 180,E1 15283.94,E2 15283.94} C_VEL
LIN {X 0,Y 346.435,Z 984.863,A -85,B 0,C 180,E1 15281.315,E2 15281.315} C_VEL
LIN {X 0,Y 346.137,Z 985.362,A -85,B 0,C 180,E1 15278.656,E2 15278.656} C_VEL
LIN {X 0,Y 346.044,Z 984.147,A -85,B 0,C 180,E1 15276.139,E2 15276.139} C_VEL
LIN {X 0,Y 346.163,Z 980.989,A -85,B 0,C 180,E1 15273.403,E2 15273.403} C_VEL
LIN {X 0,Y 346.517,Z 976.113,A -85,B 0,C 180,E1 15270.814,E2 15270.814} C_VEL
LIN {X 0,Y 347.095,Z 969.71,A -85,B 0,C 180,E1 15268.38,E2 15268.38} C_VEL
LIN {X 0,Y 347.866,Z 961.867,A -85,B 0,C 180,E1 15266.109,E2 15266.109} C_VEL
LIN {X 0,Y 348.918,Z 951.804,A -85,B 0,C 180,E1 15263.82,E2 15263.82} C_VEL
LIN {X 0,Y 350.101,Z 940.292,A -85,B 0,C 180,E1 15261.756,E2 15261.756} C_VEL
LIN {X 0,Y 351.324,Z 927.802,A -85,B 0,C 180,E1 15259.958,E2 15259.958} C_VEL
LIN {X 0,Y 352.513,Z 913.71,A -85,B 0,C 180,E1 15258.353,E2 15258.353} C_VEL
LIN {X 0,Y 353.572,Z 899.01,A -85,B 0,C 180,E1 15257.037,E2 15257.037} C_VEL
LIN {X 0,Y 354.443,Z 882.971,A -85,B 0,C 180,E1 15255.955,E2 15255.955} C_VEL
LIN {X 0,Y 354.992,Z 866.844,A -85,B 0,C 180,E1 15255.18,E2 15255.18} C_VEL
LIN {X 0,Y 355.247,Z 848.162,A -85,B 0,C 180,E1 15254.623,E2 15254.623} C_VEL
LIN {X 0,Y 358.545,Z 726.225,A -85,B 0,C 180,E1 15251.777,E2 15251.777} C_VEL
LIN {X 0,Y 357.174,Z 717.638,A -85,B 0,C 180,E1 15251.423,E2 15251.423} C_VEL
LIN {X 0,Y 358.597,Z 685.363,A -85,B 0,C 180,E1 15247.233,E2 15247.233} C_VEL
LIN {X 0,Y 358.863,Z 674.586,A -85,B 0,C 180,E1 15245.811,E2 15245.811} C_VEL
LIN {X 0,Y 354.031,Z 656.547,A -85,B 0,C 180,E1 15242.934,E2 15242.934} C_VEL
LIN {X 0,Y 348.402,Z 638.793,A -85,B 0,C 180,E1 15239.958,E2 15239.958} C_VEL
LIN {X 0,Y 345.909,Z 631.347,A -85,B 0,C 180,E1 15238.623,E2 15238.623} C_VEL
LIN {X 0,Y 345.893,Z 631.238,A -85,B 0,C 180,E1 15236.249,E2 15236.249} C_VEL
LIN {X 0,Y 347.792,Z 636.871,A -85,B 0,C 180,E1 15234.705,E2 15234.705} C_VEL
LIN {X 0,Y 352.568,Z 651.73,A -85,B 0,C 180,E1 15231.088,E2 15231.088} C_VEL
LIN {X 0,Y 356.859,Z 667.049,A -85,B 0,C 180,E1 15227.614,E2 15227.614} C_VEL
LIN {X 0,Y 359.969,Z 680.028,A -85,B 0,C 180,E1 15224.888,E2 15224.888} C_VEL
LIN {X 0,Y 357.952,Z 695.894,A -85,B 0,C 180,E1 15222.22,E2 15222.22} C_VEL
LIN {X 0,Y 364.569,Z 731.712,A -85,B 0,C 180,E1 15220.806,E2 15220.806} C_VEL
LIN {X 0,Y 363.675,Z 764.638,A -85,B 0,C 180,E1 15220.158,E2 15220.158} C_VEL
LIN {X 0,Y 362.591,Z 772.31,A -85,B 0,C 180,E1 15220.079,E2 15220.079} C_VEL
LIN {X 0,Y 356.468,Z 792.658,A -85,B 0,C 180,E1 15220.134,E2 15220.134} C_VEL
LIN {X 0,Y 355.604,Z 799.245,A -85,B 0,C 180,E1 15220.057,E2 15220.057} C_VEL
LIN {X 0,Y 354.165,Z 852.438,A -85,B 0,C 180,E1 15218.902,E2 15218.902} C_VEL
LIN {X 0,Y 353.342,Z 870.036,A -85,B 0,C 180,E1 15218.206,E2 15218.206} C_VEL
LIN {X 0,Y 352.137,Z 886.383,A -85,B 0,C 180,E1 15217.259,E2 15217.259} C_VEL
LIN {X 0,Y 350.584,Z 901.671,A -85,B 0,C 180,E1 15216.058,E2 15216.058} C_VEL
LIN {X 0,Y 348.706,Z 916.813,A -85,B 0,C 180,E1 15214.523,E2 15214.523} C_VEL
LIN {X 0,Y 346.812,Z 930.176,A -85,B 0,C 180,E1 15212.81,E2 15212.81} C_VEL
LIN {X 0,Y 344.859,Z 942.479,A -85,B 0,C 180,E1 15210.831,E2 15210.831} C_VEL
LIN {X 0,Y 343.027,Z 953.343,A -85,B 0,C 180,E1 15208.664,E2 15208.664} C_VEL
LIN {X 0,Y 341.411,Z 962.791,A -85,B 0,C 180,E1 15206.306,E2 15206.306} C_VEL
LIN {X 0,Y 340.026,Z 970.955,A -85,B 0,C 180,E1 15203.673,E2 15203.673} C_VEL
